	              // Calculate path choice
	              #tempRetValue := "LKinCtrl_CalcCircPathChoiceByIntermediatePointAndEndPoint"(circleStartPoint := #tempNextCmdIn.endPoint,
	                                                                                           circleEndPoint := #tempNextButOneCmdIn.endPoint,
	                                                                                           circleintermediatePoint := #tempNextButOneCmdIn.circleIntermediatePoint,
	                                                                                           pathPlane := #pathPlane,
	                                                                                           pathChoice => #tempNextButOneCmdIn.pathChoice);
	              
	              IF (#tempRetValue <> 0) THEN
	                #LKinCtrl_OffsetContour.returnValue := #tempRetValue;
	                #LKinCtrl_OffsetContour."region" := #COFF_REGION_TYPE_RAD_COMP_CIRC_CIRC;
	                #LKinCtrl_OffsetContour.subBlockNumber := 35058;
	                #LKinCtrl_OffsetContour.internalNumber := 431;
	                RETURN;
	              END_IF;
	              
	            ELSIF (#tempNextButOneCmdIn.circleMode = "CM_CENTER") THEN
	              // ------------ Via the circle center and the angle in a main plane ("CircMode" = 1) ------------
	              
	              // "Third" coordinate is ignored by system - also ignore here!
	              // Use start coordinate of circle instead
	              IF (#pathPlane = "CP_XZ") THEN
	                #tempNextButOneCmdIn.circleCenterPoint.y := #tempNextCmdIn.endPoint.y;
	              ELSIF (#pathPlane = "CP_YZ") THEN
	                #tempNextButOneCmdIn.circleCenterPoint.x := #tempNextCmdIn.endPoint.x;
	              ELSIF (#pathPlane = "CP_XY") THEN
	                #tempNextButOneCmdIn.circleCenterPoint.z := #tempNextCmdIn.endPoint.z;
	              END_IF;
	              
	              // Calculte correct circle end point - parameter not mandatory (and therefore probably not correct)
	              #tempRetValue := "LKinCtrl_CalcCircEndPointWithGivenCenterAndAngle"(circleStartPoint := #tempNextCmdIn.endPoint,
	                                                                                  circleCenterPoint := #tempNextButOneCmdIn.circleCenterPoint,
	                                                                                  pathPlane := #pathPlane,
	                                                                                  pathChoice := #tempNextButOneCmdIn.pathChoice,
	                                                                                  angle := #tempNextButOneCmdIn.circleAngle,
	                                                                                  endPoint => #tempNextButOneCmdIn.endPoint);
	              
	              IF (#tempRetValue <> 0) THEN
	                #LKinCtrl_OffsetContour.returnValue := #tempRetValue;
	                #LKinCtrl_OffsetContour."region" := #COFF_REGION_TYPE_RAD_COMP_CIRC_CIRC;
	                #LKinCtrl_OffsetContour.subBlockNumber := 35053;
	                #LKinCtrl_OffsetContour.internalNumber := 432;
	                RETURN;
	              END_IF;
	              
	            ELSIF (#tempNextButOneCmdIn.circleMode = "CM_RADIUS") THEN
	              // ------------ Via the circle radius and the end point in a main plane ("CircMode" = 2) ------------
	              #tempRetValue := "LKinCtrl_CalcCircCenterByRadiusAndEndPoint"(circleStartPoint := #tempNextCmdIn.endPoint,
	                                                                            circleEndPoint := #tempNextButOneCmdIn.endPoint,
	                                                                            pathPlane := #pathPlane,
	                                                                            circleRadius := #tempNextButOneCmdIn.circleRadius,
	                                                                            pathChoice := #tempNextButOneCmdIn.pathChoice,
	                                                                            circCenterPoint => #tempNextButOneCmdIn.circleCenterPoint);
	              
	              IF (#tempRetValue <> 0) THEN
	                #LKinCtrl_OffsetContour.returnValue := #tempRetValue;
	                #LKinCtrl_OffsetContour."region" := #COFF_REGION_TYPE_RAD_COMP_CIRC_CIRC;
	                #LKinCtrl_OffsetContour.subBlockNumber := 35052;
	                #LKinCtrl_OffsetContour.internalNumber := 433;
	                RETURN;
	              END_IF;
	              
	            END_IF;
	            
	            // Take care of next circular command
	            #tempRetValue := "LKinCtrl_CalcCircTangOrthPathPlane"(circlePoint := #tempNextCmdIn.endPoint,
	                                                                  circleCenterPoint := #tempNextButOneCmdIn.circleCenterPoint,
	                                                                  pathPlane := #pathPlane,
	                                                                  compDirection := #compensationDirection,
	                                                                  pathChoice := #tempNextButOneCmdIn.pathChoice,
	                                                                  vUnitTangentialPathPlane => #tempNextButOneCmdOut.tangentialUnitVecStart,
	                                                                  vUnitOrthogonalPathPlane => #tempNextButOneCmdOut.orthogonalUnitVecStart);
	            
	            IF (#tempRetValue <> 0) THEN
	              #LKinCtrl_OffsetContour.returnValue := #tempRetValue;
	              #LKinCtrl_OffsetContour."region" := #COFF_REGION_TYPE_RAD_COMP_CIRC_CIRC;
	              #LKinCtrl_OffsetContour.subBlockNumber := 35056;
	              #LKinCtrl_OffsetContour.internalNumber := 434;
	              RETURN;
	            END_IF;
	            
	            // Scale othogonal vector with tool radius to get orthogonal shift
	            #tempNextButOneCmdOut.orthogonalShiftStart := "LKinCtrl_VecScale"(vIn := #tempNextButOneCmdOut.orthogonalUnitVecStart,
	                                                                              factor := #toolRadius);
	            
	            
	            #tempNextButOneCmdOut.startPointOrthShifted := "LKinCtrl_VecAdd"(vIn1 := #tempNextCmdIn.endPoint,
	                                                                             vIn2 := #tempNextButOneCmdOut.orthogonalShiftStart);
	            
	            // ########## Intersection point of 1st circular and 2nd circular command  ##########
	            
	            IF (#tempNextCmdIn.circleMode = "CM_BORDER") THEN
	              // ------------ Via an intermediate point and the end point ("CircMode" = 0) ------------
	              // 3D circle possible
	              //
	              // Bring coordinates and parameters to same level as current point
	              #tempNextCmdStartPointOrhtShiftLevelled := #tempCurrentPointRadComp; //#tempNextCmdOut.startPointOrthShifted;
	              #tempNextCmdOut.circleCenterPoint := #tempNextCmdIn.circleCenterPoint;
	              
	              // Level parameters (third coordinate) with current point
	              CASE #pathPlane OF
	                "CP_XZ":
	                  #tempNextCmdStartPointOrhtShiftLevelled.y := #tempCurrentPoint.y;
	                  #tempNextCmdOut.circleCenterPoint.y := #tempCurrentPoint.y;
	                  
	                "CP_YZ":
	                  #tempNextCmdStartPointOrhtShiftLevelled.x := #tempCurrentPoint.x;
	                  #tempNextCmdOut.circleCenterPoint.x := #tempCurrentPoint.x;
	                  
	                "CP_XY":
	                  #tempNextCmdStartPointOrhtShiftLevelled.z := #tempCurrentPoint.z;
	                  #tempNextCmdOut.circleCenterPoint.z := #tempCurrentPoint.z;
	                ELSE
	                  #LKinCtrl_OffsetContour.returnValue := #ERR_COFF_INTERNAL;
	                  #LKinCtrl_OffsetContour."region" := #COFF_REGION_TYPE_RAD_COMP_CIRC_CIRC;
	                  #LKinCtrl_OffsetContour.internalNumber := 435;
	                  RETURN;
	              END_CASE;
	              
	              // Calculate radius of shifted 1st circle - levelled
	              #tempNextCmdOut.circleRadius := "LKinCtrl_VecAbs"("LKinCtrl_VecSub"(vIn1 := #tempNextCmdStartPointOrhtShiftLevelled,
	                                                                                                                                    vIn2 := #tempNextCmdOut.circleCenterPoint));
	            ELSE
	              #tempNextCmdOut.circleCenterPoint := #tempNextCmdIn.circleCenterPoint;
	              // Calculate radius of shifted 1st circle
	              #tempNextCmdOut.circleRadius := "LKinCtrl_VecAbs"("LKinCtrl_VecSub"(vIn1 := #tempCurrentPointRadComp,
	                                                                                                                                    vIn2 := #tempNextCmdOut.circleCenterPoint));
	            END_IF;
	            
	            IF (#tempNextButOneCmdIn.circleMode = "CM_BORDER") THEN
	              // ------------ Via an intermediate point and the end point ("CircMode" = 0) ------------
	              // 3D circle possible
	              //
	              // Bring coordinates and parameters to same level as current point
	              #tempNextButOneStartPointOrthShiftedLevelled := #tempNextButOneCmdOut.startPointOrthShifted;
	              #tempNextButOneCmdOut.circleCenterPoint := #tempNextButOneCmdIn.circleCenterPoint;
	              
	              // Level parameters (third coordinate) with current point
	              CASE #pathPlane OF
	                "CP_XZ":
	                  #tempNextButOneStartPointOrthShiftedLevelled.y := #tempCurrentPoint.y;
	                  #tempNextButOneCmdOut.circleCenterPoint.y := #tempCurrentPoint.y;
	                  
	                "CP_YZ":
	                  #tempNextButOneStartPointOrthShiftedLevelled.x := #tempCurrentPoint.x;
	                  #tempNextButOneCmdOut.circleCenterPoint.x := #tempCurrentPoint.x;
	                  
	                "CP_XY":
	                  #tempNextButOneStartPointOrthShiftedLevelled.z := #tempCurrentPoint.z;
	                  #tempNextButOneCmdOut.circleCenterPoint.z := #tempCurrentPoint.z;
	                ELSE
	                  #LKinCtrl_OffsetContour.returnValue := #ERR_COFF_INTERNAL;
	                  #LKinCtrl_OffsetContour."region" := #COFF_REGION_TYPE_RAD_COMP_CIRC_CIRC;
	                  #LKinCtrl_OffsetContour.internalNumber := 435;
	                  RETURN;
	              END_CASE;
	              // Calculate radius of shifted 2nd circle - levelled
	              #tempNextButOneCmdOut.circleRadius := "LKinCtrl_VecAbs"("LKinCtrl_VecSub"(vIn1 := #tempNextButOneStartPointOrthShiftedLevelled,
	                                                                                                                                                vIn2 := #tempNextButOneCmdOut.circleCenterPoint));
	            ELSE
	              #tempNextButOneCmdOut.circleCenterPoint := #tempNextButOneCmdIn.circleCenterPoint;
	              
	              // Calculate radius of shifted 2nd circle
	              // preliminary
	              #tempNextButOneCmdOut.circleRadius := "LKinCtrl_VecAbs"("LKinCtrl_VecSub"(vIn1 := #tempNextButOneCmdOut.startPointOrthShifted,
	                                                                                                                                                vIn2 := #tempNextButOneCmdOut.circleCenterPoint));
	            END_IF;
	            
	            // Intersection point of 1st and 2nd circle
	            #tempRetValue := "LKinCtrl_CalcCircleCircleIntersectionPoint"(circleCenterPoint1 := #tempNextCmdOut.circleCenterPoint,
	                                                                          circleCenterPoint2 := #tempNextButOneCmdOut.circleCenterPoint,
	                                                                          circleRadius1 := #tempNextCmdOut.circleRadius,
	                                                                          circleRadius2 := #tempNextButOneCmdOut.circleRadius,
	                                                                          pathPlane := #pathPlane,
	                                                                          intersectionPointA => #tempPa,
	                                                                          intersectionPointB => #tempPb);
	            IF (#tempRetValue <> 0) THEN
	              // V01.00.01
	              IF (#tempRetValue = #ERR_COFF_CIRCLE_CENTERS_EQUAL) THEN
	                // Circles are equal - use modified start point of following circle instead
	                #tempPa := #tempNextButOneCmdOut.startPointOrthShifted;
	                #tempPb := #tempNextButOneCmdOut.startPointOrthShifted;
	              ELSE
	                #LKinCtrl_OffsetContour.returnValue := #tempRetValue;
	                #LKinCtrl_OffsetContour."region" := #COFF_REGION_TYPE_RAD_COMP_CIRC_CIRC;
	                #LKinCtrl_OffsetContour.subBlockNumber := 35062;
	                #LKinCtrl_OffsetContour.internalNumber := 437;
	                RETURN;
	              END_IF;
	            END_IF;
	            
	            IF (#tempNextCmdIn.circleMode = "CM_BORDER") THEN
	              // ------------ Via an intermediate point and the end point ("CircMode" = 0) ------------
	              // 3D circle possible
	              // Relevel intersection point
	              CASE #pathPlane OF
	                "CP_XZ":
	                  #tempPa.y := #tempNextCmdIn.endPoint.y;
	                  #tempPb.y := #tempNextCmdIn.endPoint.y;
	                  
	                "CP_YZ":
	                  #tempPa.x := #tempNextCmdIn.endPoint.x;
	                  #tempPb.x := #tempNextCmdIn.endPoint.x;
	                  
	                "CP_XY":
	                  #tempPa.z := #tempNextCmdIn.endPoint.z;
	                  #tempPb.z := #tempNextCmdIn.endPoint.z;
	                ELSE
	                  #LKinCtrl_OffsetContour.returnValue := #ERR_COFF_INTERNAL;
	                  #LKinCtrl_OffsetContour."region" := #COFF_REGION_TYPE_RAD_COMP_CIRC_LIN;
	                  #LKinCtrl_OffsetContour.internalNumber := 436;
	                  RETURN;
	              END_CASE;
	            END_IF;
	            
	            // Two intersection points, use the one which is closer to the circle end point
	            #tempDistance1 := "LKinCtrl_VecAbs"("LKinCtrl_VecSub"(vIn1 := #tempNextCmdIn.endPoint, vIn2 := #tempPa));
	            #tempDistance2 := "LKinCtrl_VecAbs"("LKinCtrl_VecSub"(vIn1 := #tempNextCmdIn.endPoint, vIn2 := #tempPb));
	            
	            IF (#tempDistance1 < #tempDistance2) THEN
	              #tempNextCmdOut.endPoint := #tempPa;
	            ELSE
	              #tempNextCmdOut.endPoint := #tempPb;
	            END_IF;
	            
	          END_REGION
	          // ############# N E X T   B U T   O N E   C M D  -  N O N E #############
	        ELSE
	          REGION Next but one command NONE
	            // Output next but one coordinates - in case it's the last one
	            #tempNextButOneCmdOut.endPoint := #tempNextButOneCmdOut.endPointOrthShifted;
	            
	            // Calculate end point for circle (orthogonal shifted)
	            #tempRetValue := "LKinCtrl_CalcCircTangOrthPathPlane"(circlePoint := #tempNextCmdIn.endPoint,
	                                                                  circleCenterPoint := #tempNextCmdIn.circleCenterPoint,
	                                                                  pathPlane := #pathPlane,
	                                                                  compDirection := #compensationDirection,
	                                                                  pathChoice := #tempNextCmdIn.pathChoice,
	                                                                  vUnitTangentialPathPlane => #tempNextCmdOut.tangentialUnitVecEnd,
	                                                                  vUnitOrthogonalPathPlane => #tempNextCmdOut.orthogonalUnitVecEnd);
	            
	            IF (#tempRetValue <> 0) THEN
	              #LKinCtrl_OffsetContour.returnValue := #tempRetValue;
	              #LKinCtrl_OffsetContour."region" := #COFF_REGION_TYPE_RAD_COMP_CIRC_NONE;
	              #LKinCtrl_OffsetContour.subBlockNumber := 35056;
	              #LKinCtrl_OffsetContour.internalNumber := 450;
	              RETURN;
	            END_IF;
	            
	            // Scale othogonal vector with tool radius to get orthogonal shift
	            #tempNextCmdOut.orthogonalShiftEnd := "LKinCtrl_VecScale"(vIn := #tempNextCmdOut.orthogonalUnitVecEnd,
	                                                                      factor := #toolRadius);
	            
	            
	            #tempNextCmdOut.endPoint := "LKinCtrl_VecAdd"(vIn1 := #tempNextCmdIn.endPoint,
	                                                          vIn2 := #tempNextCmdOut.orthogonalShiftEnd);
	            (*
	            // Distinguish between different circular modes
	            IF (#tempNextCmdIn.circleMode = "CM_BORDER") THEN
	              // ------------ Via an intermediate point and the end point ("CircMode" = 0) ------------
	              
	              // Calculate end point for circle mode 0 by given mode 0
	              #tempRetValue := "LKinCtrl_CalcCircTangOrthPathPlane"(circlePoint := #tempNextCmdIn.endPoint,
	                                                                    circleCenterPoint := #tempNextCmdIn.circleCenterPoint,
	                                                                    pathPlane := #pathPlane,
	                                                                    compDirection := #compensationDirection,
	                                                                    pathChoice := #tempNextCmdIn.pathChoice,
	                                                                    vUnitTangentialPathPlane => #tempNextCmdOut.tangentialUnitVecEnd,
	                                                                    vUnitOrthogonalPathPlane => #tempNextCmdOut.orthogonalUnitVecEnd);
	              
	              IF (#tempRetValue <> 0) THEN
	                #LKinCtrl_OffsetContour.returnValue := #tempRetValue;
	                #LKinCtrl_OffsetContour."region" := #COFF_REGION_TYPE_RAD_COMP_CIRC_NONE;
	                #LKinCtrl_OffsetContour.subBlockNumber := 35056;
	                #LKinCtrl_OffsetContour.internalNumber := 450;
	                RETURN;
	              END_IF;
	              
	              // Scale othogonal vector with tool radius to get orthogonal shift
	              #tempNextCmdOut.orthogonalShiftEnd := "LKinCtrl_VecScale"(vIn := #tempNextCmdOut.orthogonalUnitVecEnd,
	                                                                        factor := #toolRadius);
	              
	              
	              #tempNextCmdOut.endPoint := "LKinCtrl_VecAdd"(vIn1 := #tempNextCmdIn.endPoint,
	                                                            vIn2 := #tempNextCmdOut.orthogonalShiftEnd);
	            ELSIF (#tempNextCmdIn.circleMode = "CM_CENTER") THEN
	              (*
	              // Calculate end point for circle mode 0 by given mode 1
	              #tempRetValue := "LKinCtrl_CalcCircEndPointWithGivenCenterAndAngle"(circleStartPoint := #tempCurrentPointRadComp,
	                                                                                  circleCenterPoint := #tempNextCmdIn.circleCenterPoint,
	                                                                                  pathPlane := #pathPlane,
	                                                                                  pathChoice := #tempNextCmdIn.pathChoice,
	                                                                                  angle := #tempNextCmdIn.circleAngle,
	                                                                                  endPoint => #tempNextCmdOut.endPoint);
	              
	              IF (#tempRetValue <> 0) THEN
	                #LKinCtrl_OffsetContour.returnValue := #tempRetValue;
	                #LKinCtrl_OffsetContour."region" := #COFF_REGION_TYPE_RAD_COMP_CIRC_NONE;
	                #LKinCtrl_OffsetContour.subBlockNumber := 35053;
	                #LKinCtrl_OffsetContour.internalNumber := 451;
	                RETURN;
	              END_IF;
	              *)
	              // Calculate end point for circle mode 0 by given mode 0
	              #tempRetValue := "LKinCtrl_CalcCircTangOrthPathPlane"(circlePoint := #tempNextCmdIn.endPoint,
	                                                                    circleCenterPoint := #tempNextCmdIn.circleCenterPoint,
	                                                                    pathPlane := #pathPlane,
	                                                                    compDirection := #compensationDirection,
	                                                                    pathChoice := #tempNextCmdIn.pathChoice,
	                                                                    vUnitTangentialPathPlane => #tempNextCmdOut.tangentialUnitVecEnd,
	                                                                    vUnitOrthogonalPathPlane => #tempNextCmdOut.orthogonalUnitVecEnd);
	              
	              IF (#tempRetValue <> 0) THEN
	                #LKinCtrl_OffsetContour.returnValue := #tempRetValue;
	                #LKinCtrl_OffsetContour."region" := #COFF_REGION_TYPE_RAD_COMP_CIRC_NONE;
	                #LKinCtrl_OffsetContour.subBlockNumber := 35056;
	                #LKinCtrl_OffsetContour.internalNumber := 450;
	                RETURN;
	              END_IF;
	              
	              // Scale othogonal vector with tool radius to get orthogonal shift
	              #tempNextCmdOut.orthogonalShiftEnd := "LKinCtrl_VecScale"(vIn := #tempNextCmdOut.orthogonalUnitVecEnd,
	                                                                        factor := #toolRadius);
	              
	              
	              #tempNextCmdOut.endPoint := "LKinCtrl_VecAdd"(vIn1 := #tempNextCmdIn.endPoint,
	                                                            vIn2 := #tempNextCmdOut.orthogonalShiftEnd);
	              
	            ELSIF (#tempNextCmdIn.circleMode = "CM_RADIUS") THEN
	              (*
	              // ------------ Via the circle radius and the end point in a main plane ("CircMode" = 2) ------------
	              // Calculate angle between center/start and center/end of circle - always the smaller one!!!
	              #tempRetValue := "LKinCtrl_CalcAngleBetweenVectors"(point1 := #tempCurrentPointRadComp,//#tempNextCmdOut.startPointOrthShifted,
	                                                                  point2 := #tempNextCmdIn.endPoint,//#tempNextCmdOut.endPoint,
	                                                                  intersectionPoint := #tempNextCmdIn.circleCenterPoint,
	                                                                  angle => #tempAngle);
	              
	              IF (#tempRetValue <> 0) THEN
	                #LKinCtrl_OffsetContour.returnValue := #tempRetValue;
	                #LKinCtrl_OffsetContour."region" := #COFF_REGION_TYPE_RAD_COMP_CIRC_NONE;
	                #LKinCtrl_OffsetContour.subBlockNumber := 35059;
	                #LKinCtrl_OffsetContour.internalNumber := 452;
	                RETURN;
	              END_IF;
	              
	              // Calculate end point for circle mode 0 by given mode 2
	              #tempRetValue := "LKinCtrl_CalcCircEndPointWithGivenCenterAndAngle"(circleStartPoint := #tempCurrentPointRadComp, //tempNextCmdOut.startPointOrthShifted,
	                                                                                  circleCenterPoint := #tempNextCmdIn.circleCenterPoint,
	                                                                                  pathPlane := #pathPlane,
	                                                                                  pathChoice := #tempNextCmdIn.pathChoice,
	                                                                                  angle := #tempAngle,
	                                                                                  endPoint => #tempNextCmdOut.endPoint);
	              
	              
	              
	              IF (#tempRetValue <> 0) THEN
	                #LKinCtrl_OffsetContour.returnValue := #tempRetValue;
	                #LKinCtrl_OffsetContour."region" := #COFF_REGION_TYPE_RAD_COMP_CIRC_NONE;
	                #LKinCtrl_OffsetContour.subBlockNumber := 35053;
	                #LKinCtrl_OffsetContour.internalNumber := 453;
	                RETURN;
	              END_IF;
	              *)
	              ;
	            END_IF;
	            *)
	            
	          END_REGION
	        END_IF;
	        
	        
	        // ############# M O D I F Y   N E X T   C I R C U L A R   C O M M A N D   #############
	        REGION Modify next circular command
	          // Distinguish between different circular modes
	          IF (#tempNextCmdIn.circleMode = "CM_BORDER") THEN
	            
	            // ------------ Via an intermediate point and the end point ("CircMode" = 0) ------------
	            // Calculate intermediate point for circle mode 0 by given mode 0
	            // Calculate circle paramters
	            #tempRetValue := "LKinCtrl_CalcCircTangOrthPathPlane"(circlePoint := #tempNextCmdIn.circleIntermediatePoint,
	                                                                  circleCenterPoint := #tempNextCmdIn.circleCenterPoint,
	                                                                  pathPlane := #pathPlane,
	                                                                  compDirection := #compensationDirection,
	                                                                  pathChoice := #tempNextCmdIn.pathChoice,
	                                                                  vUnitTangentialPathPlane => #tempNextCmdOut.tangentialUnitVecIntermediate,
	                                                                  vUnitOrthogonalPathPlane => #tempNextCmdOut.orthogonalUnitVecIntermediate);
	            
	            IF (#tempRetValue <> 0) THEN
	              #LKinCtrl_OffsetContour.returnValue := #tempRetValue;
	              #LKinCtrl_OffsetContour."region" := #COFF_REGION_TYPE_RAD_COMP_CIRC_GEN;
	              #LKinCtrl_OffsetContour.subBlockNumber := 35056;
	              #LKinCtrl_OffsetContour.internalNumber := 460;
	              RETURN;
	            END_IF;
	            
	            // Scale othogonal vector with tool radius to get orthogonal shift
	            #tempNextCmdOut.orthogonalShiftIntermediate := "LKinCtrl_VecScale"(vIn := #tempNextCmdOut.orthogonalUnitVecIntermediate,
	                                                                               factor := #toolRadius);
	            
	            
	            #tempNextCmdOut.circleIntermediatePoint := "LKinCtrl_VecAdd"(vIn1 := #tempNextCmdIn.circleIntermediatePoint,
	                                                                         vIn2 := #tempNextCmdOut.orthogonalShiftIntermediate);
	            
	            // Change circle mode to 0 - intermediate point and the end point ("CircMode" = 0)
	            #tempNextCmdOut.circleMode := "CM_BORDER";
	            
	          ELSIF (#tempNextCmdIn.circleMode = "CM_CENTER") THEN
	            
	            // Take care of greater angles
	            // #tempMod := TRUNC(#tempNextCmdIn.circleAngle / 180.0);
	            // IF (#tempMod >= 3) THEN
	            //   #tempAngle := #tempNextCmdIn.circleAngle - ((#tempMod - 1) * 180);
	            // ELSE
	            //   #tempAngle := #tempNextCmdIn.circleAngle;
	            // END_IF;
	            
	            // V01.02.02
	            // Calculate compensated angle
	            #tempRetValue := "LKinCtrl_CalcAngleBetweenVectors"(point1 := #tempCurrentPointRadComp, //tempNextCmdOut.startPointOrthShifted,
	                                                                point2 := #tempNextCmdOut.endPoint,
	                                                                intersectionPoint := #tempNextCmdIn.circleCenterPoint,
	                                                                angle => #tempAngle);
	            
	            IF (#tempRetValue <> 0) THEN
	              #LKinCtrl_OffsetContour.returnValue := #tempRetValue;
	              #LKinCtrl_OffsetContour."region" := #COFF_REGION_TYPE_RAD_COMP_CIRC_GEN;
	              #LKinCtrl_OffsetContour.subBlockNumber := 35059;
	              #LKinCtrl_OffsetContour.internalNumber := 461;
	              RETURN;
	            END_IF;
	            //
	            // Calculate intermediate point for circle mode 0 by given mode 1
	            #tempRetValue := "LKinCtrl_CalcCircEndPointWithGivenCenterAndAngle"(circleStartPoint := #tempCurrentPointRadComp, // tempNextCmdOut.startPointOrthShifted,
	                                                                                circleCenterPoint := #tempNextCmdIn.circleCenterPoint,
	                                                                                pathPlane := #pathPlane,
	                                                                                pathChoice := #tempNextCmdIn.pathChoice,
	                                                                                angle := #tempAngle / 2.0,//(#tempNextCmdIn.circleAngle / 2.0),
	                                                                                endPoint => #tempNextCmdOut.circleIntermediatePoint);
	            IF (#tempRetValue <> 0) THEN
	              #LKinCtrl_OffsetContour.returnValue := #tempRetValue;
	              #LKinCtrl_OffsetContour."region" := #COFF_REGION_TYPE_RAD_COMP_CIRC_GEN;
	              #LKinCtrl_OffsetContour.subBlockNumber := 35053;
	              #LKinCtrl_OffsetContour.internalNumber := 462;
	              RETURN;
	            END_IF;
	            
	            // Ceck if resulting path choice (circle with intermediate point) has changed --> circle larger than 360°
	            // Calculate path choice
	            #tempRetValue := "LKinCtrl_CalcCircPathChoiceByIntermediatePointAndEndPoint"(circleStartPoint := #tempCurrentPointRadComp, //tempNextCmdOut.startPointOrthShifted,
	                                                                                         circleEndPoint := #tempNextCmdOut.endPoint,
	                                                                                         circleintermediatePoint := #tempNextCmdOut.circleIntermediatePoint,
	                                                                                         pathPlane := #pathPlane,
	                                                                                         pathChoice => #tempPathChoice);
	            
	            
	            IF (#tempRetValue <> 0) THEN
	              #LKinCtrl_OffsetContour.returnValue := #tempRetValue;
	              #LKinCtrl_OffsetContour."region" := #COFF_REGION_TYPE_RAD_COMP_CIRC_GEN;
	              #LKinCtrl_OffsetContour.subBlockNumber := 35058;
	              #LKinCtrl_OffsetContour.internalNumber := 463;
	              RETURN;
	            END_IF;
	            
	            IF ((#tempNextCmdIn.pathChoice <> #tempPathChoice) OR
	              (#tempNextCmdIn.circleAngle >= 360.0))
	            THEN
	              
	              // V01.02.02 - done before now
	              // // Calculate additional angle between center/start and center/end of circle - always the smaller one!!!
	              // #tempRetValue := "LKinCtrl_CalcAngleBetweenVectors"(point1 := #tempCurrentPointRadComp, //tempNextCmdOut.startPointOrthShifted,
	              //                                                     point2 := #tempNextCmdOut.endPoint,
	              //                                                     intersectionPoint := #tempNextCmdIn.circleCenterPoint,
	              //                                                     angle => #tempAngle);
	              
	              // IF (#tempRetValue <> 0) THEN
	              //   #LKinCtrl_OffsetContour.returnValue := #tempRetValue;
	              //   #LKinCtrl_OffsetContour."region" := #COFF_REGION_TYPE_RAD_COMP_CIRC_GEN;
	              //   #LKinCtrl_OffsetContour.subBlockNumber := 35059;
	              //   #LKinCtrl_OffsetContour.internalNumber := 463;
	              //   RETURN;
	              // END_IF;
	              
	              // Circle > 360° - not possible with circle type border
	              IF (#tempNextCmdIn.pathChoice <> #tempPathChoice) THEN
	                #tempNextCmdOut.circleAngle := (TRUNC((#tempNextCmdIn.circleAngle + 180.0) / 360.0) * 360.0) + #tempAngle;
	              ELSE
	                #tempNextCmdOut.circleAngle := (TRUNC((#tempNextCmdIn.circleAngle + 180.0) / 360.0) * 360.0) - #tempAngle;
	              END_IF;
	              
	              #tempNextCmdOut.circleMode := "CM_CENTER";
	            ELSE
	              
	              // V01.02.02
	              // Output angle - for debugging only
	              #tempNextCmdOut.circleAngle := #tempAngle;
	              
	              // Change circle mode to 0 - intermediate point and the end point ("CircMode" = 0)
	              #tempNextCmdOut.circleMode := "CM_BORDER";
	            END_IF;
	            
	          ELSIF (#tempNextCmdIn.circleMode = "CM_RADIUS") THEN
	            // ------------ Via the circle radius and the end point in a main plane ("CircMode" = 2) ------------
	            // Calculate angle between center/start and center/end of circle - always the smaller one!!!
	            #tempRetValue := "LKinCtrl_CalcAngleBetweenVectors"(point1 := #tempCurrentPointRadComp,
	                                                                point2 := #tempNextCmdOut.endPoint,
	                                                                intersectionPoint := #tempNextCmdIn.circleCenterPoint,
	                                                                angle => #tempAngle);
	            
	            IF (#tempRetValue <> 0) THEN
	              #LKinCtrl_OffsetContour.returnValue := #tempRetValue;
	              #LKinCtrl_OffsetContour."region" := #COFF_REGION_TYPE_RAD_COMP_CIRC_GEN;
	              #LKinCtrl_OffsetContour.subBlockNumber := 35059;
	              #LKinCtrl_OffsetContour.internalNumber := 464;
	              RETURN;
	            END_IF;
	            
	            // Calculate intermediate point for circle mode 0 by given mode 2
	            #tempRetValue := "LKinCtrl_CalcCircEndPointWithGivenCenterAndAngle"(circleStartPoint := #tempCurrentPointRadComp, //tempNextCmdOut.startPointOrthShifted,
	                                                                                circleCenterPoint := #tempNextCmdIn.circleCenterPoint,
	                                                                                pathPlane := #pathPlane,
	                                                                                pathChoice := #tempNextCmdIn.pathChoice,
	                                                                                angle := (#tempAngle / 2.0),
	                                                                                endPoint => #tempNextCmdOut.circleIntermediatePoint);
	            
	            IF (#tempRetValue <> 0) THEN
	              #LKinCtrl_OffsetContour.returnValue := #tempRetValue;
	              #LKinCtrl_OffsetContour."region" := #COFF_REGION_TYPE_RAD_COMP_CIRC_GEN;
	              #LKinCtrl_OffsetContour.subBlockNumber := 35053;
	              #LKinCtrl_OffsetContour.internalNumber := 465;
	              RETURN;
	            END_IF;
	            
	            // Change circle mode to 0 - intermediate point and the end point ("CircMode" = 0)
	            #tempNextCmdOut.circleMode := "CM_BORDER";
	            
	          END_IF;
	          
	          // Additional check - has the direction between start - end and start - compensated end changed
	          // --> Reversal path with "small" length (and "large" tool radius) leads to unexpected circle (mathematical correct but in an unexpected direction)
	          REGION Additional plausibility check
	            #tempRetValue := "LKinCtrl_CalcAngleBetweenVectors"(point1 := #tempNextCmdOut.endPoint,
	                                                                point2 := #tempNextCmdIn.endPoint,
	                                                                intersectionPoint := #tempCurrentPoint,
	                                                                angle => #tempAngle);
	            
	            IF (#tempRetValue <> 0) THEN
	              #LKinCtrl_OffsetContour.returnValue := #tempRetValue;
	              #LKinCtrl_OffsetContour."region" := #COFF_REGION_TYPE_RAD_COMP_CIRC_GEN;
	              #LKinCtrl_OffsetContour.subBlockNumber := 35059;
	              #LKinCtrl_OffsetContour.internalNumber := 470;
	              RETURN;
	            END_IF;
	            
	            IF ((#tempAngle > #COFF_CIRC_REVERSAL_TOLERANCE_ANGLE) AND
	              ("LKinCtrl_VecAbs"("LKinCtrl_VecSub"(vIn1 := #tempNextCmdOut.endPoint,
	                                                                      vIn2 := #tempNextCmdOut.circleIntermediatePoint)) < (2.0 * #toolRadius)))
	            THEN
	              #LKinCtrl_OffsetContour.returnValue := #ERR_COFF_NO_SOLUTION_FOR_GIVEN_CIRCULAR_CMD;
	              #LKinCtrl_OffsetContour."region" := #COFF_REGION_TYPE_RAD_COMP_CIRC_GEN;
	              #LKinCtrl_OffsetContour.subBlockNumber := 0;
	              #LKinCtrl_OffsetContour.internalNumber := 471;
	              RETURN;
	            END_IF;
	            
	          END_REGION
	          
	          // V01.02.02
	          REGION Additional plausibility check
	            // Check if circle radius has become smaller than possible - compensation inside
	            
	            // Calculate the length end point circle center 
	            #tempRetValue := "LKinCtrl_CalcVecDistancePathPlane"(vectorInA := #tempNextCmdIn.endPoint,
	                                                                 vectorInB := #tempNextCmdIn.circleCenterPoint,
	                                                                 pathPlane := #pathPlane,
	                                                                 distancePathPlane => #tempCircleDistance1);
	            
	            IF (#tempRetValue <> 0) THEN
	              #LKinCtrl_OffsetContour.returnValue := #tempRetValue;
	              #LKinCtrl_OffsetContour."region" := #COFF_REGION_TYPE_RAD_COMP_CIRC_GEN;
	              #LKinCtrl_OffsetContour.subBlockNumber := 35067;
	              #LKinCtrl_OffsetContour.internalNumber := 472;
	              RETURN;
	            END_IF;
	            
	            #tempRetValue := "LKinCtrl_CalcVecDistancePathPlane"(vectorInA := #tempNextCmdOut.endPoint,
	                                                                 vectorInB := #tempNextCmdIn.circleCenterPoint,
	                                                                 pathPlane := #pathPlane,
	                                                                 distancePathPlane => #tempCircleDistance2);
	            
	            IF (#tempRetValue <> 0) THEN
	              #LKinCtrl_OffsetContour.returnValue := #tempRetValue;
	              #LKinCtrl_OffsetContour."region" := #COFF_REGION_TYPE_RAD_COMP_CIRC_GEN;
	              #LKinCtrl_OffsetContour.subBlockNumber := 35067;
	              #LKinCtrl_OffsetContour.internalNumber := 473;
	              RETURN;
	            END_IF;
	            
	            IF (#tempCircleDistance2 < #tempCircleDistance1) THEN
	              // inside circle - check plausibility
	              // Tool radius must not be greater than circle radius
	              IF (#toolRadius > (#tempCircleDistance1 - #RADIUS_PLAUSIBLITY_TOLERANCE)) THEN
	                #LKinCtrl_OffsetContour.returnValue := #ERR_COFF_NO_SOLUTION_FOR_GIVEN_CIRCULAR_CMD;
	                #LKinCtrl_OffsetContour."region" := #COFF_REGION_TYPE_RAD_COMP_CIRC_GEN;
	                #LKinCtrl_OffsetContour.subBlockNumber := 0;
	                #LKinCtrl_OffsetContour.internalNumber := 474;
	                RETURN;
	              END_IF;
	              // Tool radius must not be greater than circle start and end point (uncompensated)
	              #tempRetValue := "LKinCtrl_CalcVecDistancePathPlane"(vectorInA := #tempCurrentPoint,
	                                                                   vectorInB := #tempNextCmdIn.endPoint,
	                                                                   pathPlane := #pathPlane,
	                                                                   distancePathPlane => #tempCircleDistance3);
	              
	              IF (#tempRetValue <> 0) THEN
	                #LKinCtrl_OffsetContour.returnValue := #tempRetValue;
	                #LKinCtrl_OffsetContour."region" := #COFF_REGION_TYPE_RAD_COMP_CIRC_GEN;
	                #LKinCtrl_OffsetContour.subBlockNumber := 35067;
	                #LKinCtrl_OffsetContour.internalNumber := 475;
	                RETURN;
	              END_IF;
	              
	              IF (#toolRadius > (#tempCircleDistance3 - #RADIUS_PLAUSIBLITY_TOLERANCE)) THEN
	                #LKinCtrl_OffsetContour.returnValue := #ERR_COFF_NO_SOLUTION_FOR_GIVEN_CIRCULAR_CMD;
	                #LKinCtrl_OffsetContour."region" := #COFF_REGION_TYPE_RAD_COMP_CIRC_GEN;
	                #LKinCtrl_OffsetContour.subBlockNumber := 0;
	                #LKinCtrl_OffsetContour.internalNumber := 476;
	                RETURN;
	              END_IF;
	              
	            END_IF;
	            
	          END_REGION
	        END_REGION
	      END_IF;
	    END_REGION
	    
	  END_IF;
	  
	  // V01.00.01
	  // Output before length compensation
	  #nextPositionAbsoluteRadCompOut := "LKinCtrl_3DPointToCartesianCoord"(#tempNextCmdOut.endPoint);
	END_REGION TOOL_RADIUS_COMPENSATION
	
	// Tool length compensation
	REGION TOOL_LENGTH_COMPENSATION
	  IF (#tempToolLengthComp) THEN
	    // Next command
	    // -------------------------------------------------------------------------------------
	    // Compensate coordinates of according to path plane
	    // End point
	    #tempRetValue := "LKinCtrl_CalcToolLengthCompensation"(toolLength := #toolLength,
	                                                           pathPlane := #pathPlane,
	                                                           point := #tempNextCmdOut.endPoint);
	    IF (#tempRetValue <> 0) THEN
	      #LKinCtrl_OffsetContour.returnValue := #tempRetValue;
	      #LKinCtrl_OffsetContour."region" := #COFF_REGION_TYPE_LEN_COMP_NEXT;
	      #LKinCtrl_OffsetContour.subBlockNumber := 35070;
	      #LKinCtrl_OffsetContour.internalNumber := 601;
	      RETURN;
	    END_IF;
	    
	    // Circle coordinates
	    IF (#tempNextCmdOut.cmdType = "LKINCTRL_MC_MOVECIRCULARABS") THEN
	      
	      IF (#tempNextCmdOut.circleMode = "CM_BORDER") THEN
	        
	        #tempRetValue := "LKinCtrl_CalcToolLengthCompensation"(toolLength := #toolLength,
	                                                               pathPlane := #pathPlane,
	                                                               point := #tempNextCmdOut.circleIntermediatePoint);
	        IF (#tempRetValue <> 0) THEN
	          #LKinCtrl_OffsetContour.returnValue := #tempRetValue;
	          #LKinCtrl_OffsetContour."region" := #COFF_REGION_TYPE_LEN_COMP_NEXT;
	          #LKinCtrl_OffsetContour.subBlockNumber := 35070;
	          #LKinCtrl_OffsetContour.internalNumber := 602;
	          RETURN;
	        END_IF;
	        
	      ELSIF (#tempNextCmdOut.circleMode = "CM_CENTER") THEN
	        
	        #tempRetValue := "LKinCtrl_CalcToolLengthCompensation"(toolLength := #toolLength,
	                                                               pathPlane := #pathPlane,
	                                                               point := #tempNextCmdOut.circleCenterPoint);
	        IF (#tempRetValue <> 0) THEN
	          #LKinCtrl_OffsetContour.returnValue := #tempRetValue;
	          #LKinCtrl_OffsetContour."region" := #COFF_REGION_TYPE_LEN_COMP_NEXT;
	          #LKinCtrl_OffsetContour.subBlockNumber := 35070;
	          #LKinCtrl_OffsetContour.internalNumber := 603;
	          RETURN;
	        END_IF;
	        
	      ELSIF (#tempNextCmdOut.circleMode = "CM_RADIUS") THEN
	        ;
	      ELSE
	        #LKinCtrl_OffsetContour.returnValue := #ERR_COFF_INTERNAL; // Internal error
	        #LKinCtrl_OffsetContour."region" := #COFF_REGION_TYPE_LEN_COMP_NEXT;
	        #LKinCtrl_OffsetContour.internalNumber := 604;
	        RETURN;
	      END_IF;
	    END_IF;
	    
	    // Intermediate command
	    // -------------------------------------------------------------------------------------
	    // Compensate coordinates of according to path plane
	    IF (#tempIntermediateCmdOut.cmdType <> -1) THEN
	      
	      // End point
	      #tempRetValue := "LKinCtrl_CalcToolLengthCompensation"(toolLength := #toolLength,
	                                                             pathPlane := #pathPlane,
	                                                             point := #tempIntermediateCmdOut.endPoint);
	      IF (#tempRetValue <> 0) THEN
	        #LKinCtrl_OffsetContour.returnValue := #tempRetValue;
	        #LKinCtrl_OffsetContour."region" := #COFF_REGION_TYPE_LEN_COMP_INTER_CMD;
	        #LKinCtrl_OffsetContour.subBlockNumber := 35070;
	        #LKinCtrl_OffsetContour.internalNumber := 605;
	        RETURN;
	      END_IF;
	      
	      // Always circle by intemdiate point and end point
	      #tempRetValue := "LKinCtrl_CalcToolLengthCompensation"(toolLength := #toolLength,
	                                                             pathPlane := #pathPlane,
	                                                             point := #tempIntermediateCmdOut.circleIntermediatePoint);
	      IF (#tempRetValue <> 0) THEN
	        #LKinCtrl_OffsetContour.returnValue := #tempRetValue;
	        #LKinCtrl_OffsetContour."region" := #COFF_REGION_TYPE_LEN_COMP_INTER_CMD;
	        #LKinCtrl_OffsetContour.subBlockNumber := 35070;
	        #LKinCtrl_OffsetContour.internalNumber := 606;
	        RETURN;
	      END_IF;
	    END_IF;
	    
	    // Next but one command - not needed - no output
	    // -------------------------------------------------------------------------------------
	    (*
	    // Compensate coordinates of according to path plane
	    // End point
	    #tempRetValue := "LKinCtrl_CalcToolLengthCompensation"(toolLength := #toolLength,
	                                                           pathPlane := #pathPlane,
	                                                           point := #tempNextButOneCmdOut.endPoint);
	    IF (#tempRetValue <> 0) THEN
	      #LKinCtrl_OffsetContour.returnValue := #tempRetValue;
	      #LKinCtrl_OffsetContour."region" := #COFF_REGION_TYPE_LEN_COMP_NEXT_BUT_ONE_CMD;
	      #LKinCtrl_OffsetContour.subBlockNumber := 35070;
	      #LKinCtrl_OffsetContour.internalNumber := 607
	      RETURN;
	    END_IF;
	    *)
	  END_IF;
	END_REGION
	
	REGION Output data
	  
	  // ############# O U T P U T   D A T A  #############
	  // ###################################### 
	  IF (#tempToolRadiusComp OR #tempToolLengthComp) THEN
	    // Next command
	    
	    #nextCommandOut.cmdType := #tempNextCmdOut.cmdType;
	    #nextCommandOut.cmdCoordinates.cartesianPosition := "LKinCtrl_3DPointToCartesianCoord"(#tempNextCmdOut.endPoint);
	    
	    IF (#tempNextCmdOut.cmdType = "LKINCTRL_MC_MOVECIRCULARABS") THEN
	      #nextCommandOut.cmdParameters.circleParameters.circMode := #tempNextCmdOut.circleMode;
	      
	      IF (#tempNextCmdOut.circleMode = "CM_BORDER") THEN
	        #nextCommandOut.cmdParameters.circleParameters.auxPoint[1] := #tempNextCmdOut.circleIntermediatePoint.x;
	        #nextCommandOut.cmdParameters.circleParameters.auxPoint[2] := #tempNextCmdOut.circleIntermediatePoint.y;
	        #nextCommandOut.cmdParameters.circleParameters.auxPoint[3] := #tempNextCmdOut.circleIntermediatePoint.z;
	        // *** AW 2022-05-29 - debugging only - compensated angle
	        #nextCommandOut.cmdParameters.circleParameters.arc := #tempNextCmdOut.circleAngle;
	        
	      ELSIF (#tempNextCmdOut.circleMode = "CM_CENTER") THEN
	        #nextCommandOut.cmdParameters.circleParameters.pathChoice := #tempNextCmdIn.pathChoice;
	        #nextCommandOut.cmdParameters.circleParameters.circlePlane := #tempNextCmdIn.circlePlane;
	        #nextCommandOut.cmdParameters.circleParameters.auxPoint[1] := #tempNextCmdOut.circleCenterPoint.x;
	        #nextCommandOut.cmdParameters.circleParameters.auxPoint[2] := #tempNextCmdOut.circleCenterPoint.y;
	        #nextCommandOut.cmdParameters.circleParameters.auxPoint[3] := #tempNextCmdOut.circleCenterPoint.z;
	        #nextCommandOut.cmdParameters.circleParameters.arc := #tempNextCmdOut.circleAngle; // #tempNextCmdIn.circleAngle;
	        
	      ELSIF (#tempNextCmdOut.circleMode = "CM_RADIUS") THEN
	        #nextCommandOut.cmdParameters.circleParameters.pathChoice := #tempNextCmdIn.pathChoice;
	        #nextCommandOut.cmdParameters.circleParameters.circlePlane := #tempNextCmdIn.circlePlane;
	        #nextCommandOut.cmdParameters.circleParameters.radius := #tempNextCmdIn.circleRadius;
	        
	      ELSE
	        #LKinCtrl_OffsetContour.returnValue := #ERR_COFF_INTERNAL; // Internal error
	        #LKinCtrl_OffsetContour."region" := #COFF_REGION_TYPE_OUTPUT_DATA;
	        RETURN;
	      END_IF;
	    END_IF;
	    
	    // Coordinate a
	    // ------------
	    // Linear absolute
	    IF (#tempNextCmdIn.cmdType = "LKINCTRL_MC_MOVELINEARABS") THEN
	      // Absolute coordinates
	      #nextCommandOut.cmdCoordinates.cartesianPosition.a := #nextCommandIn.cmdCoordinates.cartesianPosition.a;
	      // Linear relative
	    ELSIF (#tempNextCmdIn.cmdType = "LKINCTRL_MC_MOVELINEARREL") THEN
	      // Relative coordinates -> calculate absolute coordinate (always)
	      #nextCommandOut.cmdCoordinates.cartesianPosition.a := #currentPosIn.positionAbsolute.a + #nextCommandIn.cmdCoordinates.cartesianPosition.a;
	      // Circular absolute  
	    ELSIF (#tempNextCmdIn.cmdType = "LKINCTRL_MC_MOVECIRCULARABS") THEN
	      // Absolute coordinates
	      #nextCommandOut.cmdCoordinates.cartesianPosition.a := #nextCommandIn.cmdCoordinates.cartesianPosition.a;
	      // Circular relative  
	    ELSIF (#tempNextCmdIn.cmdType = "LKINCTRL_MC_MOVECIRCULARREL") THEN
	      // Relative coordinates -> calculate absolute coordinate (always)
	      #nextCommandOut.cmdCoordinates.cartesianPosition.a := #currentPosIn.positionAbsolute.a + #nextCommandIn.cmdCoordinates.cartesianPosition.a;
	    END_IF;
	    
	    // Output absolute end point for next cycle (including coordinate a)
	    #nextPositionAbsoluteOut := "LKinCtrl_3DPointToCartesianCoord"(#tempNextCmdIn.endPoint);
	    #nextPositionAbsoluteOut.a := #nextCommandOut.cmdCoordinates.cartesianPosition.a;
	    
	    // Output absolute end point (radius compensated) for next cycle (including coordinate a)
	    // V01.00.01
	    // nextPositionAbsoluteRadCompOut := "LKinCtrl_3DPointToCartesianCoord"(#tempNextCmdOut.endPoint);
	    #nextPositionAbsoluteRadCompOut.a := #nextCommandOut.cmdCoordinates.cartesianPosition.a;
	    
	    // Intermediate command
	    IF (#tempIntermediateCmdOut.cmdType <> -1) THEN
	      
	      // Take all parameter preliminary
	      #intermediateCommandOut := #nextCommandIn;
	      
	      #intermediateCommandOut.cmdType := #tempIntermediateCmdOut.cmdType;
	      #intermediateCommandOut.cmdParameters.circleParameters.circMode := #tempIntermediateCmdOut.circleMode;
	      
	      // Circle by intemdiate point and end point
	      #intermediateCommandOut.cmdCoordinates.cartesianPosition := "LKinCtrl_3DPointToCartesianCoord"(#tempIntermediateCmdOut.endPoint);
	      #intermediateCommandOut.cmdParameters.circleParameters.auxPoint[1] := #tempIntermediateCmdOut.circleIntermediatePoint.x;
	      #intermediateCommandOut.cmdParameters.circleParameters.auxPoint[2] := #tempIntermediateCmdOut.circleIntermediatePoint.y;
	      #intermediateCommandOut.cmdParameters.circleParameters.auxPoint[3] := #tempIntermediateCmdOut.circleIntermediatePoint.z;
	      
	      // Coordinate a
	      #intermediateCommandOut.cmdCoordinates.cartesianPosition.a := #nextCommandOut.cmdCoordinates.cartesianPosition.a;
	    ELSE
	      #intermediateCommandOut.cmdType := -1;
	    END_IF;
	    
	    // Next but one command
	    //nextButOneCommandOut.cmdType := #tempNextButOneCmdIn.cmdType;
	    //nextButOneCommandOut.cmdCoordinates.cartesianPosition := "LKinCtrl_3DPointToCartesianCoord"(#tempNextButOneCmdOut.endPoint);
	    #nextButOneCommandOut.transitionParameter[1] := #tempNextButOneCmdOut.transitionParameter1;
	  ELSE
	    // Next command
	    #nextCommandOut := #nextCommandIn;
	  END_IF;
	  
	END_REGION
	
	#LKinCtrl_OffsetContour.returnValue := 16#0;
	#LKinCtrl_OffsetContour."region" := #COFF_REGION_TYPE_NONE;
	#LKinCtrl_OffsetContour.subBlockNumber := 16#0;
	#LKinCtrl_OffsetContour.internalNumber := 0;
	
	
END_FUNCTION

FUNCTION "LKinCtrl_CartesianCoordTo3DPoint" : "LKinCtrl_typeCOff3DPoint"
TITLE = LKinCtrl_CartesianCoordTo3DPoint
{ S7_Optimized_Access := 'TRUE' }
AUTHOR : 'handling.team.automation@siemens.com'
FAMILY : LKinCtrl
VERSION : 5.0
//The function converts data type "LKinCtrl_typeCartesianPosition" in "LKinCtrl_typeCOff3DPoint"
   VAR_INPUT 
      cartesianCoord : "LKinCtrl_typeCartesianPosition";   // Cartesian input coordinate
   END_VAR


BEGIN
	//==========================================================================================
	// SIEMENS AG
	// (c)Copyright 2019 All Rights Reserved
	//------------------------------------------------------------------------------------------
	// Library: LCOffset
	// Tested with: S7-1515T-3 PN/DP
	// Engineering: TIA Portal V15
	// Restrictions: ---
	// Requirements: S7-1500T FW 2.5
	// Functionality: The function converts data type "LKinCtrl_typeCartesianPosition" in "LKinCtrl_typeCOff3DPoint"
	// Support: tech.team.motioncontrol@siemens.com
	// Note: Parameter comments are only available in language 'English (United States)'
	//------------------------------------------------------------------------------------------
	// Change log table:
	// Version    Date          Expert in charge    Changes applied
	// 01.00.00   2019-02-14    AW                  created
	//===========================================================================================
	//
	#LKinCtrl_CartesianCoordTo3DPoint.x := #cartesianCoord.x;
	#LKinCtrl_CartesianCoordTo3DPoint.y := #cartesianCoord.y;
	#LKinCtrl_CartesianCoordTo3DPoint.z := #cartesianCoord.z;
END_FUNCTION

FUNCTION "LKinCtrl_VecAdd" : "LKinCtrl_typeCOff3DPoint"
TITLE = LKinCtrl_VecAdd
{ S7_Optimized_Access := 'TRUE' }
AUTHOR : 'handling.team.automation@siemens.com'
FAMILY : LKinCtrl
VERSION : 5.0
//Add two coordinates (X, Y, Z) of "LKinCtrl_typeCOff3DPoint"
   VAR_INPUT 
      vIn1 : "LKinCtrl_typeCOff3DPoint";   // Input vector 1
      vIn2 : "LKinCtrl_typeCOff3DPoint";   // Input vector 2
   END_VAR


BEGIN
	//=============================================================================
	// SIEMENS AG
	// (c)Copyright 2018 All Rights Reserved
	//-----------------------------------------------------------------------------
	// Library: - 
	// Tested with: S7-1516T-3 PN
	// Engineering: TIA Portal V15
	// Restrictions: -
	// Requirements: S7-1500/S7-1500T FW 2.5
	// Functionality: Add two coordinates (X, Y, Z) of "LKinCtrl_typeCOff3DPoint"
	//-----------------------------------------------------------------------------
	// Change log table:
	// Version  Date       Expert in charge Changes applied
	// 01.00.00 2018-10-26 AW               created
	//=============================================================================
	#LKinCtrl_VecAdd.x := #vIn1.x + #vIn2.x;
	#LKinCtrl_VecAdd.y := #vIn1.y + #vIn2.y;
	#LKinCtrl_VecAdd.z := #vIn1.z + #vIn2.z;
END_FUNCTION

FUNCTION "LKinCtrl_VecAbs" : LReal
TITLE = LKinCtrl_VecAbs
{ S7_Optimized_Access := 'TRUE' }
AUTHOR : 'handling.team.automation@siemens.com'
FAMILY : LKinCtrl
VERSION : 5.0
//Calculate length of vector of coordinates (X, Y, Z) of "LKinCtrl_typeCOff3DPoint"
   VAR_INPUT 
      vIn : "LKinCtrl_typeCOff3DPoint";   // Input vector
   END_VAR


BEGIN
	//=============================================================================
	// SIEMENS AG
	// (c)Copyright 2018 All Rights Reserved
	//-----------------------------------------------------------------------------
	// Library: - 
	// Tested with: S7-1516T-3 PN
	// Engineering: TIA Portal V15
	// Restrictions: -
	// Requirements: S7-1500/S7-1500T FW 2.5
	// Functionality: Calculate length of vector of coordinates (X, Y, Z) of "LKinCtrl_typeCOff3DPoint"
	//-----------------------------------------------------------------------------
	// Change log table:
	// Version  Date       Expert in charge Changes applied
	// 01.00.00 2018-10-26 AW               created
	//=============================================================================
	
	#LKinCtrl_VecAbs := SQRT(#vIn.x * #vIn.x + #vIn.y * #vIn.y + #vIn.z * #vIn.z);
END_FUNCTION

FUNCTION "LKinCtrl_VecSub" : "LKinCtrl_typeCOff3DPoint"
TITLE = LKinCtrl_VecSub
{ S7_Optimized_Access := 'TRUE' }
AUTHOR : 'handling.team.automation@siemens.com'
FAMILY : LKinCtrl
VERSION : 5.0
//Substract two coordinates (X, Y, Z) of "LKinCtrl_typeCOff3DPoint"
   VAR_INPUT 
      vIn1 : "LKinCtrl_typeCOff3DPoint";   // Input vector 1
      vIn2 : "LKinCtrl_typeCOff3DPoint";   // Input vector 2
   END_VAR


BEGIN
	//=============================================================================
	// SIEMENS AG
	// (c)Copyright 2018 All Rights Reserved
	//-----------------------------------------------------------------------------
	// Library: - 
	// Tested with: S7-1516T-3 PN
	// Engineering: TIA Portal V15
	// Restrictions: -
	// Requirements: S7-1500/S7-1500T FW 2.5
	// Functionality: Substract two coordinates (X, Y, Z) of "LKinCtrl_typeCOff3DPoint"
	//-----------------------------------------------------------------------------
	// Change log table:
	// Version  Date       Expert in charge Changes applied
	// 01.00.00 2018-10-26 AW               created
	//=============================================================================
	#LKinCtrl_VecSub.x := #vIn1.x - #vIn2.x;
	#LKinCtrl_VecSub.y := #vIn1.y - #vIn2.y;
	#LKinCtrl_VecSub.z := #vIn1.z - #vIn2.z;
	
	
END_FUNCTION

FUNCTION "LKinCtrl_CalcVecDistancePathPlane" : Word
TITLE = LKinCtrl_CalcVecDistancePathPlane
{ S7_Optimized_Access := 'TRUE' }
AUTHOR : 'handling.team.automation@siemens.com'
FAMILY : LKinCtrl
VERSION : 5.0
//Calculate vector distance with respect to path plane
   VAR_INPUT 
      vectorInA : "LKinCtrl_typeCOff3DPoint";   // Vector A
      vectorInB : "LKinCtrl_typeCOff3DPoint";   // vector B
      pathPlane : Int;   // Path plane: XZ= 0, YZ=1, XY= 2
   END_VAR

   VAR_OUTPUT 
      distancePathPlane : LReal;   // Distance with respect to path plane
   END_VAR

   VAR_TEMP 
      tempVectorA : "LKinCtrl_typeCOff3DPoint";
      tempVectorB : "LKinCtrl_typeCOff3DPoint";
   END_VAR

   VAR CONSTANT 
      ERR_COFF_INVALID_PATH_PLANE : Word := 16#8303;   // Error - invalid path plane
   END_VAR


BEGIN
	//=============================================================================
	// SIEMENS AG
	// (c)Copyright 2019 All Rights Reserved
	//-----------------------------------------------------------------------------
	// Library: - 
	// Tested with: S7-1516T-3 PN
	// Engineering: TIA Portal V15
	// Restrictions: -
	// Requirements: S7-1500/S7-1500T FW 2.5
	// Functionality: Calculate vector distance with respect to path plane
	//-----------------------------------------------------------------------------
	// Change log table:
	// Version  Date       Expert in charge Changes applied
	// 01.00.00 2019-02-15 AW               created
	//=============================================================================
	REGION PLAUSIBILITY_CHECK
	  // Check path plane
	  IF ((#pathPlane >= "CP_XZ") AND (#pathPlane <= "CP_XY"))
	  THEN
	    ;
	  ELSE
	    #LKinCtrl_CalcVecDistancePathPlane := #ERR_COFF_INVALID_PATH_PLANE; // Invalid path plane
	    RETURN;
	  END_IF;
	END_REGION PLAUSIBILITY_CHECK
	
	
	REGION CALCULATION
	  #tempVectorA := #vectorInA;
	  #tempVectorB := #vectorInB;
	  
	  // Eleminate "third" coordinate
	  CASE #pathPlane OF
	    "CP_XY":
	      #tempVectorA.z := 0.0;
	      #tempVectorB.z := 0.0;
	      
	    "CP_XZ":
	      #tempVectorA.y := 0.0;
	      #tempVectorB.y := 0.0;
	      
	    "CP_YZ":
	      #tempVectorA.x := 0.0;
	      #tempVectorB.x := 0.0;
	  END_CASE;
	
	  #distancePathPlane := "LKinCtrl_VecAbs"("LKinCtrl_VecSub"(vIn1:=#tempVectorB, vIn2:=#tempVectorA));
	  
	  
	  
	END_REGION CALCULATION
	
	#LKinCtrl_CalcVecDistancePathPlane := 0; // o.k.
END_FUNCTION

FUNCTION "LKinCtrl_CalcCircEndPointWithGivenCenterAndAngle" : Word
TITLE = LKinCtrl_CalcCircEndPointWithGivenCenterAndAngle
{ S7_Optimized_Access := 'TRUE' }
AUTHOR : 'handling.team.automation@siemens.com'
FAMILY : LKinCtrl
VERSION : 5.0
//Calculate circle end point with given start point, circle center and angle
   VAR_INPUT 
      circleStartPoint : "LKinCtrl_typeCOff3DPoint";   // Circle start point
      circleCenterPoint : "LKinCtrl_typeCOff3DPoint";   // Circle center point
      pathPlane : Int;   // Path plane: XZ= 0, YZ=1, XY= 2
      pathChoice : DInt;   // Circle path choice: positive= 0, negative= 1
      angle : LReal;   // Circle angle
   END_VAR

   VAR_OUTPUT 
      endPoint : "LKinCtrl_typeCOff3DPoint";
   END_VAR

   VAR_TEMP 
      tempSin : LReal;
      tempCos : LReal;
      tempVOrthogonal : "LKinCtrl_typeCOff3DPoint";   // Othogonal vector
      tempVRotated : "LKinCtrl_typeCOff3DPoint";
   END_VAR

   VAR CONSTANT 
      ERR_COFF_INVALID_PATH_PLANE : Word := 16#8303;   // Error - invalid path plane
      ERR_COFF_INVALID_COMPENSATION_DIRECTION : Word := 16#8304;   // Error - invalid compensation direction
   END_VAR


BEGIN
	//=============================================================================
	// SIEMENS AG
	// (c)Copyright 2019 All Rights Reserved
	//-----------------------------------------------------------------------------
	// Library: - 
	// Tested with: S7-1516T-3 PN
	// Engineering: TIA Portal V15
	// Restrictions: -
	// Requirements: S7-1500/S7-1500T FW 2.5
	// Functionality: Calculate circle end point with given
	// start point, circle center and angle
	//-----------------------------------------------------------------------------
	// Change log table:
	// Version  Date       Expert in charge Changes applied
	// 01.00.00 2019-01-24 AW               created
	//=============================================================================
	
	REGION PLAUSIBILITY_CHECK
	  // Check path plane
	  IF ((#pathPlane >= "CP_XZ") AND (#pathPlane <= "CP_XY"))
	  THEN
	    // Check compensation direction
	    IF ((#pathChoice >= 0) AND (#pathChoice <= 1))
	    THEN
	      ;
	    ELSE
	      #LKinCtrl_CalcCircEndPointWithGivenCenterAndAngle := #ERR_COFF_INVALID_COMPENSATION_DIRECTION; // Invalid compensation direction
	      RETURN;
	    END_IF;
	  ELSE
	    #LKinCtrl_CalcCircEndPointWithGivenCenterAndAngle := #ERR_COFF_INVALID_PATH_PLANE; // Invalid path plane
	    RETURN;
	  END_IF;
	END_REGION PLAUSIBILITY_CHECK
	
	REGION CALCULATION
	  
	// Calc radius vector (difference vector) circle center to start point
	#tempVOrthogonal := "LKinCtrl_VecSub"(vIn1 := #circleStartPoint, vIn2 := #circleCenterPoint);
	
	IF (#pathChoice = 0) THEN
	  // positive
	  #tempSin := SIN(#angle * "LKINCTRL_PI" / 180.0);
	  #tempCos := COS(#angle * "LKINCTRL_PI" / 180.0);
	ELSE
	  #tempSin := SIN(- #angle * "LKINCTRL_PI" / 180.0);
	  #tempCos := COS(- #angle * "LKINCTRL_PI" / 180.0);
	END_IF;
	
	// Check path plane
	IF (#pathPlane = "CP_XY") THEN
	  // Rotation around Z
	  #tempVRotated.x := #tempVOrthogonal.x * #tempCos - #tempVOrthogonal.y * #tempSin;      // Calculation X
	  #tempVRotated.y := #tempVOrthogonal.x * #tempSin + #tempVOrthogonal.y * #tempCos;      // Calculation Y
	  #tempVRotated.z := #tempVOrthogonal.z;                                                 // Calculation Z
	  
	ELSIF (#pathPlane = "CP_XZ") THEN
	  // Rotation around Y
	  #tempVRotated.x := #tempVOrthogonal.x * #tempCos + #tempVOrthogonal.z * #tempSin;      // Calculation X
	  #tempVRotated.y := #tempVOrthogonal.y;                                                 // Calculation Y
	  #tempVRotated.z := -#tempVOrthogonal.x * #tempSin + #tempVOrthogonal.z * #tempCos;     // Calculation Z
	  
	ELSIF (#pathPlane = "CP_YZ") THEN
	  // Rotation around X
	  #tempVRotated.x := #tempVOrthogonal.x;      // Calculation X
	  #tempVRotated.y := #tempVOrthogonal.y * #tempCos - #tempVOrthogonal.z * #tempSin;       // Calculation Y
	  #tempVRotated.z := #tempVOrthogonal.y * #tempSin + #tempVOrthogonal.z * #tempCos;     // Calculation Z
	END_IF;
	
	// Calculate end point of circle by adding the rotated vector to the circle center point
	#endPoint := "LKinCtrl_VecAdd"(vIn1:=#tempVRotated, vIn2:=#circleCenterPoint);
	
	END_REGION CALCULATION
	
	#LKinCtrl_CalcCircEndPointWithGivenCenterAndAngle := 0;
END_FUNCTION

FUNCTION "LKinCtrl_CalcLineTangOrthPathPlane" : Word
TITLE = LKinCtrl_CalcLineTangOrthPathPlane
{ S7_Optimized_Access := 'TRUE' }
AUTHOR : 'handling.team.automation@siemens.com'
FAMILY : LKinCtrl
VERSION : 5.0
//Calculate orthogonal and tangential vector of a line with respect ot the path plane
   VAR_INPUT 
      pathPlane : Int;   // Path plane: XZ= 0, YZ=1, XY= 2
      compDirection : Int;   // Tool radius compensation direction: left=1, right = 0
      vInFirst : "LKinCtrl_typeCOff3DPoint";   // Next position
      vInSecond : "LKinCtrl_typeCOff3DPoint";   // Current position
   END_VAR

   VAR_OUTPUT 
      vUnitTangentialPathPlane : "LKinCtrl_typeCOff3DPoint";   // Output tangential vector - path plane - unit vector
      vUnitOrthogonalPathPlane : "LKinCtrl_typeCOff3DPoint";   // Output orthogonal vector - path plane - unit vector
   END_VAR

   VAR_TEMP 
      tempVOrthogonal : "LKinCtrl_typeCOff3DPoint";   // Othogonal vector
      tempVTangential : "LKinCtrl_typeCOff3DPoint";   // Tangential vector
   END_VAR

   VAR CONSTANT 
      ERR_COFF_INVALID_PATH_PLANE : Word := 16#8303;   // Error - invalid path plane
      ERR_COFF_INVALID_COMPENSATION_DIRECTION : Word := 16#8304;   // Error - invalid compensation direction
   END_VAR


BEGIN
	//=============================================================================
	// SIEMENS AG
	// (c)Copyright 2019 All Rights Reserved
	//-----------------------------------------------------------------------------
	// Library: - 
	// Tested with: S7-1516T-3 PN
	// Engineering: TIA Portal V15
	// Restrictions: -
	// Requirements: S7-1500/S7-1500T FW 2.5
	// Functionality: Calculate orthogonal and tangential vector of a line
	// with respect ot the path plane
	//-----------------------------------------------------------------------------
	// Change log table:
	// Version  Date       Expert in charge Changes applied
	// 01.00.00 2019-02-05 AW               created
	//=============================================================================
	
	REGION PLAUSIBILITY_CHECK
	// Check path plane
	  IF ((#pathPlane >= "CP_XZ") AND (#pathPlane <= "CP_XY"))
	THEN
	  // Check compensation direction
	  IF ((#compDirection >= "LKINCTRL_COMP_LEFT") AND (#compDirection <= "LKINCTRL_COMP_RIGHT"))
	  THEN
	    ;
	  ELSE
	    #LKinCtrl_CalcLineTangOrthPathPlane := #ERR_COFF_INVALID_COMPENSATION_DIRECTION; // Invalid compensation direction
	    RETURN;
	  END_IF;
	ELSE
	  #LKinCtrl_CalcLineTangOrthPathPlane := #ERR_COFF_INVALID_PATH_PLANE; // Invalid path plane
	  RETURN;
	END_IF;
	
	END_REGION PLAUSIBILITY_CHECK
	
	REGION CALCULATION
	  // Calculate difference vector (take care of path plane) - tangential vector
	  #tempVTangential := "LKinCtrl_VecSub"(vIn1 := #vInFirst,
	                                        vIn2 := #vInSecond);
	  
	  // Take care of path plane
	  CASE #pathPlane OF
	    "CP_XY":
	      #tempVTangential.z := 0.0;
	      
	    "CP_XZ":
	      #tempVTangential.y := 0.0;
	      
	    "CP_YZ":
	      #tempVTangential.x := 0.0;
	  END_CASE;
	  
	  // Normalize vector
	  #tempVTangential := "LKinCtrl_VecUnit"(vIn := #tempVTangential);
	  
	  
	// Calculate orthogonal vector to current vector depending on path plane and compensation direction
	CASE #pathPlane OF
	  "CP_XY":
	    IF (#compDirection = "LKINCTRL_COMP_LEFT") THEN
	      #tempVOrthogonal.x := - #tempVTangential.y;
	      #tempVOrthogonal.y := #tempVTangential.x;
	      #tempVOrthogonal.z := 0.0;
	    ELSE
	      #tempVOrthogonal.x := #tempVTangential.y;
	      #tempVOrthogonal.y := - #tempVTangential.x;
	      #tempVOrthogonal.z := 0.0;          
	    END_IF;
	    
	  "CP_XZ":
	    (*
	    IF (#compDirection = "LKINCTRL_COMP_LEFT") THEN
	      #tempVOrthogonal.x := #tempVTangential.z;
	      #tempVOrthogonal.y := 0.0;
	      #tempVOrthogonal.z := - #tempVTangential.x;
	    ELSE
	      #tempVOrthogonal.x := - #tempVTangential.z;
	      #tempVOrthogonal.y := 0.0;
	      #tempVOrthogonal.z := #tempVTangential.x;
	    END_IF;*)
	    
	    IF (#compDirection = "LKINCTRL_COMP_LEFT") THEN
	      #tempVOrthogonal.x := -#tempVTangential.z;
	      #tempVOrthogonal.y := 0.0;
	      #tempVOrthogonal.z := #tempVTangential.x;
	    ELSE
	      #tempVOrthogonal.x := #tempVTangential.z;
	      #tempVOrthogonal.y := 0.0;
	      #tempVOrthogonal.z := -#tempVTangential.x;
	    END_IF;
	    
	  "CP_YZ":
	    IF (#compDirection = "LKINCTRL_COMP_LEFT") THEN
	      #tempVOrthogonal.x := 0.0;
	      #tempVOrthogonal.y := - #tempVTangential.z;
	      #tempVOrthogonal.z := #tempVTangential.y;
	    ELSE
	      #tempVOrthogonal.x := 0.0;
	      #tempVOrthogonal.y := #tempVTangential.z;
	      #tempVOrthogonal.z := - #tempVTangential.y;
	    END_IF;
	END_CASE;
	END_REGION CALCULATION
	
	#vUnitTangentialPathPlane := #tempVTangential;
	#vUnitOrthogonalPathPlane := #tempVOrthogonal;
	#LKinCtrl_CalcLineTangOrthPathPlane := 0;
	
	
	
END_FUNCTION

FUNCTION "LKinCtrl_VecUnit" : "LKinCtrl_typeCOff3DPoint"
TITLE = LKinCtrl_VecUnit
{ S7_Optimized_Access := 'TRUE' }
AUTHOR : 'handling.team.automation@siemens.com'
FAMILY : LKinCtrl
VERSION : 5.0
//Create unit vector of coordinates (X, Y, Z) of "LKinCtrl_typeCOff3DPoint"
   VAR_INPUT 
      vIn : "LKinCtrl_typeCOff3DPoint";   // Input vector
   END_VAR


BEGIN
	//=============================================================================
	// SIEMENS AG
	// (c)Copyright 2018 All Rights Reserved
	//-----------------------------------------------------------------------------
	// Library: - 
	// Tested with: S7-1516T-3 PN
	// Engineering: TIA Portal V15
	// Restrictions: -
	// Requirements: S7-1500/S7-1500T FW 2.5
	// Functionality: Create unit vector of coordinates (X, Y, Z) of "LKinCtrl_typeCOff3DPoint"
	//-----------------------------------------------------------------------------
	// Change log table:
	// Version  Date       Expert in charge Changes applied
	// 01.00.00 2018-08-27 SF               created
	//=============================================================================
	
	//Out = In/abs(In)
	#LKinCtrl_VecUnit := "LKinCtrl_VecDivScal"(vIn := #vIn,
	                                           sIn := "LKinCtrl_VecAbs"(#vIn));
	
	
END_FUNCTION

FUNCTION "LKinCtrl_VecDivScal" : "LKinCtrl_typeCOff3DPoint"
TITLE = LKinCtrl_VecDivScal
{ S7_Optimized_Access := 'TRUE' }
AUTHOR : 'handling.team.automation@siemens.com'
FAMILY : LKinCtrl
VERSION : 5.0
//Divide coordinate with scalar of coordinates (X, Y, Z) of "LKinCtrl_typeCOff3DPoint"
   VAR_INPUT 
      vIn : "LKinCtrl_typeCOff3DPoint";   // Input vector
      sIn : LReal;   // Input scalar
   END_VAR


BEGIN
	//=============================================================================
	// SIEMENS AG
	// (c)Copyright 2018 All Rights Reserved
	//-----------------------------------------------------------------------------
	// Library: - 
	// Tested with: S7-1516T-3 PN
	// Engineering: TIA Portal V15
	// Restrictions: -
	// Requirements: S7-1500/S7-1500T FW 2.5
	// Functionality: Divide coordinate with scalar of coordinates (X, Y, Z) of "LKinCtrl_typeCOff3DPoint"
	//-----------------------------------------------------------------------------
	// Change log table:
	// Version  Date       Expert in charge Changes applied
	// 01.00.00 2018-10-26 AW               created
	//=============================================================================
	
	IF (#sIn <> 0.0) THEN
	  #LKinCtrl_VecDivScal.x := #vIn.x / #sIn;
	  #LKinCtrl_VecDivScal.y := #vIn.y / #sIn;
	  #LKinCtrl_VecDivScal.z := #vIn.z / #sIn;
	ELSE
	  #LKinCtrl_VecDivScal.x := 0.0;
	  #LKinCtrl_VecDivScal.y := 0.0;
	  #LKinCtrl_VecDivScal.z := 0.0;
	END_IF;
END_FUNCTION

FUNCTION "LKinCtrl_VecScale" : "LKinCtrl_typeCOff3DPoint"
TITLE = LKinCtrl_VecScale
{ S7_Optimized_Access := 'TRUE' }
AUTHOR : 'handling.team.automation@siemens.com'
FAMILY : LKinCtrl
VERSION : 5.0
//Scale vector (X, Y, Z) of "LKinCtrl_typeCOff3DPoint"
   VAR_INPUT 
      vIn : "LKinCtrl_typeCOff3DPoint";   // Input vector
      factor : LReal;   // Scaling factor
   END_VAR


BEGIN
	//=============================================================================
	// SIEMENS AG
	// (c)Copyright 2018 All Rights Reserved
	//-----------------------------------------------------------------------------
	// Library: - 
	// Tested with: S7-1516T-3 PN
	// Engineering: TIA Portal V15
	// Restrictions: -
	// Requirements: S7-1500/S7-1500T FW 2.5
	// Functionality: Scale vector (X, Y, Z) of "LKinCtrl_typeCOff3DPoint"
	//-----------------------------------------------------------------------------
	// Change log table:
	// Version  Date       Expert in charge Changes applied
	// 01.00.00 2018-10-26 AW               created
	//=============================================================================
	
	#LKinCtrl_VecScale.x := #vIn.x * #factor;
	#LKinCtrl_VecScale.y := #vIn.y * #factor;
	#LKinCtrl_VecScale.z := #vIn.z * #factor;
	
END_FUNCTION

FUNCTION "LKinCtrl_CalcLineLineIntersectionPoint" : Word
TITLE = LKinCtrl_CalcLineLineIntersectionPoint
{ S7_Optimized_Access := 'TRUE' }
AUTHOR : 'handling.team.automation@siemens.com'
FAMILY : LKinCtrl
VERSION : 5.0
//Calculate the line segment Pa/Pb that is the shortest route between two lines P1P2 and P3P4
   VAR_INPUT 
      startPointFirstLine : "LKinCtrl_typeCOff3DPoint";   // Start point first line
      endPointFirstLine : "LKinCtrl_typeCOff3DPoint";   // End point first line
      startPointSecondLine : "LKinCtrl_typeCOff3DPoint";   // Start point second line
      endPointSecondLine : "LKinCtrl_typeCOff3DPoint";   // End point second line
   END_VAR

   VAR_OUTPUT 
      intersectionPointA : "LKinCtrl_typeCOff3DPoint";   // Intersection point a
      intersectionPointB : "LKinCtrl_typeCOff3DPoint";   // Intersection point b
      muA : LReal;   // Direction vector a
      muB : LReal;   // Direction vector b
   END_VAR

   VAR_TEMP 
      tempP13 : "LKinCtrl_typeCOff3DPoint";
      tempP43 : "LKinCtrl_typeCOff3DPoint";
      tempP21 : "LKinCtrl_typeCOff3DPoint";
      tempD1343 : LReal;
      tempD4321 : LReal;
      tempD1321 : LReal;
      tempD4343 : LReal;
      tempD2121 : LReal;
      tempNumer : LReal;
      tempDenom : LReal;
   END_VAR

   VAR CONSTANT 
      COFF_EPS : LReal := 0.001;   // Internal constant
      ERR_COFF_LINES_DO_NOT_INTERSECT : Word := 16#8312;   // Error - no solution, lines don't intersect
      ERR_COFF_ZERO_VECTOR : Word := 16#8313;   // Error - zero vector
   END_VAR


BEGIN
	//=============================================================================
	// SIEMENS AG
	// (c)Copyright 2019 All Rights Reserved
	//-----------------------------------------------------------------------------
	// Library: - 
	// Tested with: S7-1516T-3 PN
	// Engineering: TIA Portal V15
	// Restrictions: -
	// Requirements: S7-1500/S7-1500T FW 2.5
	// Functionality: Calculate the line segment Pa/Pb that is the shortest route
	// between two lines P1P2 and P3P4. Calculate also the values of mua and mub where
	// Pa = P1 + mua (P2 - P1)
	// Pb = P3 + mub (P4 - P3)
	// Return error if the lines don't intersect
	//-----------------------------------------------------------------------------
	// Change log table:
	// Version  Date       Expert in charge Changes applied
	// 01.00.00 2019-02-05 AW               created
	//=============================================================================
	REGION PLAUSIBILITY_CHECK
	
	END_REGION PLAUSIBILITY_CHECK
	
	REGION CALCULATION
	  #tempP13.x := #startPointFirstLine.x - #startPointSecondLine.x;
	  #tempP13.y := #startPointFirstLine.y - #startPointSecondLine.y;
	  #tempP13.z := #startPointFirstLine.z - #startPointSecondLine.z;
	  #tempP43.x := #endPointSecondLine.x - #startPointSecondLine.x;
	  #tempP43.y := #endPointSecondLine.y - #startPointSecondLine.y;
	  #tempP43.z := #endPointSecondLine.z - #startPointSecondLine.z;
	  IF ((ABS(#tempP43.x) < #COFF_EPS) AND (ABS(#tempP43.y) < #COFF_EPS) AND (ABS(#tempP43.z) < #COFF_EPS)) THEN
	    #LKinCtrl_CalcLineLineIntersectionPoint := #ERR_COFF_LINES_DO_NOT_INTERSECT;
	    RETURN;
	  END_IF;
	  
	  #tempP21.x := #endPointFirstLine.x - #startPointFirstLine.x;
	  #tempP21.y := #endPointFirstLine.y - #startPointFirstLine.y;
	  #tempP21.z := #endPointFirstLine.z - #startPointFirstLine.z;
	  IF ((ABS(#tempP21.x) < #COFF_EPS) AND (ABS(#tempP21.y) < #COFF_EPS) AND (ABS(#tempP21.z) < #COFF_EPS)) THEN
	    #LKinCtrl_CalcLineLineIntersectionPoint := #ERR_COFF_LINES_DO_NOT_INTERSECT;
	    RETURN;
	  END_IF;
	  
	  #tempD1343 := #tempP13.x * #tempP43.x + #tempP13.y * #tempP43.y + #tempP13.z * #tempP43.z;
	  #tempD4321 := #tempP43.x * #tempP21.x + #tempP43.y * #tempP21.y + #tempP43.z * #tempP21.z;
	  #tempD1321 := #tempP13.x * #tempP21.x + #tempP13.y * #tempP21.y + #tempP13.z * #tempP21.z;
	  #tempD4343 := #tempP43.x * #tempP43.x + #tempP43.y * #tempP43.y + #tempP43.z * #tempP43.z;
	  #tempD2121 := #tempP21.x * #tempP21.x + #tempP21.y * #tempP21.y + #tempP21.z * #tempP21.z;
	  
	  #tempDenom := #tempD2121 * #tempD4343 - #tempD4321 * #tempD4321;
	  IF (ABS(#tempDenom) < #COFF_EPS) THEN
	    #LKinCtrl_CalcLineLineIntersectionPoint := #ERR_COFF_LINES_DO_NOT_INTERSECT;
	    RETURN;
	  END_IF;
	  
	  #tempNumer := #tempD1343 * #tempD4321 - #tempD1321 * #tempD4343;
	  
	  #muA := #tempNumer / #tempDenom;
	  #muB := (#tempD1343 + #tempD4321 * #muA) / #tempD4343;
	  
	  #intersectionPointA.x := #startPointFirstLine.x + #muA * #tempP21.x;
	  #intersectionPointA.y := #startPointFirstLine.y + #muA * #tempP21.y;
	  #intersectionPointA.z := #startPointFirstLine.z + #muA * #tempP21.z;
	
	  #intersectionPointB.x := #startPointSecondLine.x + #muB * #tempP43.x;
	  #intersectionPointB.y := #startPointSecondLine.y + #muB * #tempP43.y;
	  #intersectionPointB.z := #startPointSecondLine.z + #muB * #tempP43.z;
	  
	END_REGION
	#LKinCtrl_CalcLineLineIntersectionPoint := 0;
END_FUNCTION

FUNCTION "LKinCtrl_CheckInnerOuterCorner" : Word
TITLE = LKinCtrl_CheckInnerOuterCorner
{ S7_Optimized_Access := 'TRUE' }
AUTHOR : 'handling.team.automation@siemens.com'
FAMILY : LKinCtrl
VERSION : 5.0
//Check for inner or outer corner
   VAR_INPUT 
      vInFirst : "LKinCtrl_typeCOff3DPoint";   // Input vector first
      vInSecond : "LKinCtrl_typeCOff3DPoint";   // Input vector second
      pathPlane : Int;   // Path plane: XZ= 0, YZ=1, XY= 2
      direction : Int;   // Tool radius compensation direction: left=1, right = 0
   END_VAR

   VAR_OUTPUT 
      cornerType : Int;   // Corner type - 0: outer corner, 1: inner corner
   END_VAR

   VAR_TEMP 
      tempCrossVec : "LKinCtrl_typeCOff3DPoint";
   END_VAR

   VAR CONSTANT 
      ERR_COFF_INVALID_PATH_PLANE : Word := 16#8303;   // Invalid path plane
      ERR_COFF_INVALID_COMPENSATION_DIRECTION : Word := 16#8304;   // Invalid compensation direction
   END_VAR


BEGIN
	//=============================================================================
	// SIEMENS AG
	// (c)Copyright 2019 All Rights Reserved
	//-----------------------------------------------------------------------------
	// Library: - 
	// Tested with: S7-1516T-3 PN
	// Engineering: TIA Portal V15
	// Restrictions: -
	// Requirements: S7-1500/S7-1500T FW 2.5
	// Functionality: Check for inner or outer corner
	//-----------------------------------------------------------------------------
	// Change log table:
	// Version  Date       Expert in charge Changes applied
	// 01.00.00 2019-01-24 AW               created
	// 01.00.01 2020-10-13 AW               bugfix - path plane CP_XZ - different orientation, not against third axis!
	//=============================================================================
	REGION PLAUSIBILITY_CHECK
	  // Check path plane
	  IF ((#pathPlane >= "CP_XZ") AND (#pathPlane <= "CP_XY"))
	  THEN
	    // Check compensation direction
	    IF ((#direction >= "LKINCTRL_COMP_LEFT") AND (#direction <= "LKINCTRL_COMP_RIGHT"))
	    THEN
	      ;
	    ELSE
	      #LKinCtrl_CheckInnerOuterCorner := #ERR_COFF_INVALID_COMPENSATION_DIRECTION; // Invalid compensation direction
	      RETURN;
	    END_IF;
	  ELSE
	    #LKinCtrl_CheckInnerOuterCorner := #ERR_COFF_INVALID_PATH_PLANE; // Invalid path plane
	    RETURN;
	  END_IF;
	END_REGION PLAUSIBILITY_CHECK
	
	REGION CALCULATION
	  #tempCrossVec := "LKinCtrl_VecCrossProd"(vIn1 := #vInFirst,
	                                           vIn2 := #vInSecond);
	  
	// Check path plane
	IF (#pathPlane = "CP_XY") THEN
	  IF (#direction = "LKINCTRL_COMP_RIGHT") THEN
	    IF (#tempCrossVec.z > 0.0) THEN
	      #cornerType := "LKINCTRL_OUTER_CORNER";
	    ELSE
	      #cornerType := "LKINCTRL_INNER_CORNER";
	    END_IF;
	  ELSE
	    IF (#tempCrossVec.z < 0.0) THEN
	      #cornerType := "LKINCTRL_OUTER_CORNER";
	    ELSE
	      #cornerType := "LKINCTRL_INNER_CORNER";
	    END_IF;
	  END_IF;
	  
	// 2020-10-13 AW path plane CP_XZ - different orientation, not against third axis!
	// direction changed
	ELSIF (#pathPlane = "CP_XZ") THEN
	    IF (#direction = "LKINCTRL_COMP_RIGHT") THEN
	      IF (#tempCrossVec.y > 0.0) THEN
	        #cornerType := "LKINCTRL_INNER_CORNER";
	      ELSE
	        #cornerType := "LKINCTRL_OUTER_CORNER";
	      END_IF;
	    ELSE
	      IF (#tempCrossVec.y < 0.0) THEN
	        #cornerType := "LKINCTRL_INNER_CORNER";
	      ELSE
	        #cornerType := "LKINCTRL_OUTER_CORNER";
	      END_IF;
	    END_IF;
	  ELSIF (#pathPlane = "CP_YZ") THEN
	  IF (#direction = "LKINCTRL_COMP_RIGHT") THEN
	    IF (#tempCrossVec.x > 0.0) THEN
	      #cornerType := "LKINCTRL_OUTER_CORNER";
	    ELSE
	      #cornerType := "LKINCTRL_INNER_CORNER";
	    END_IF;
	  ELSE
	    IF (#tempCrossVec.x < 0.0) THEN
	      #cornerType := "LKINCTRL_OUTER_CORNER";
	    ELSE
	      #cornerType := "LKINCTRL_INNER_CORNER";
	    END_IF;
	  END_IF;
	END_IF;
	
	#LKinCtrl_CheckInnerOuterCorner := 0;
	END_REGION CALCULATION
END_FUNCTION

FUNCTION "LKinCtrl_VecCrossProd" : "LKinCtrl_typeCOff3DPoint"
TITLE = LKinCtrl_VecCrossProd
{ S7_Optimized_Access := 'TRUE' }
AUTHOR : 'handling.team.automation@siemens.com'
FAMILY : LKinCtrl
VERSION : 5.0
//Cross product of two coordinates (X, Y, Z) of "LKinCtrl_typeCOff3DPoint"
   VAR_INPUT 
      vIn1 : "LKinCtrl_typeCOff3DPoint";   // Input vector 1
      vIn2 : "LKinCtrl_typeCOff3DPoint";   // Input vector 2
   END_VAR


BEGIN
	//=============================================================================
	// SIEMENS AG
	// (c)Copyright 2018 All Rights Reserved
	//-----------------------------------------------------------------------------
	// Library: - 
	// Tested with: S7-1516T-3 PN
	// Engineering: TIA Portal V15
	// Restrictions: -
	// Requirements: S7-1500/S7-1500T FW 2.5
	// Functionality: Cross product of two coordinates (X, Y, Z) of "LKinCtrl_typeCOff3DPoint"
	//-----------------------------------------------------------------------------
	// Change log table:
	// Version  Date       Expert in charge Changes applied
	// 01.00.00 2019-01-24 AW               created
	//=============================================================================
	
	#LKinCtrl_VecCrossProd.x := #vIn1.y * #vIn2.z - #vIn1.z * #vIn2.y;
	#LKinCtrl_VecCrossProd.y := #vIn1.z * #vIn2.x - #vIn1.x * #vIn2.z;
	#LKinCtrl_VecCrossProd.z := #vIn1.x * #vIn2.y - #vIn1.y * #vIn2.x;
	
	
END_FUNCTION

FUNCTION "LKinCtrl_CalcCircleIntermediatePos" : Void
TITLE = LKinCtrl_CalcCircleIntermediatePos
{ S7_Optimized_Access := 'TRUE' }
AUTHOR : 'handling.team.automation@siemens.com'
FAMILY : LKinCtrl
VERSION : 5.0
//Calculate intermediate point of circle with given initial end point, calculated end point and tool radius
   VAR_INPUT 
      initialEndPoint : "LKinCtrl_typeCOff3DPoint";   // Initial end point
      newEndPoint : "LKinCtrl_typeCOff3DPoint";   // New calculated end point
      toolRadius : LReal;   // Tool radius
   END_VAR

   VAR_OUTPUT 
      circIntermediatePoint : "LKinCtrl_typeCOff3DPoint";   // circle intermediate point
   END_VAR

   VAR_TEMP 
      tempVecDiff : "LKinCtrl_typeCOff3DPoint";
      tempUnitVecDiff : "LKinCtrl_typeCOff3DPoint";
   END_VAR


BEGIN
	//=============================================================================
	// SIEMENS AG
	// (c)Copyright 2019 All Rights Reserved
	//-----------------------------------------------------------------------------
	// Library: - 
	// Tested with: S7-1516T-3 PN
	// Engineering: TIA Portal V15
	// Restrictions: -
	// Requirements: S7-1500/S7-1500T FW 2.5
	// Functionality: Calculate intermediate point of circle
	// with given initial end point, calculated end point and tool radius
	//-----------------------------------------------------------------------------
	// Change log table:
	// Version  Date       Expert in charge Changes applied
	// 01.00.00 2019-02-05 AW               created
	//=============================================================================
	
	REGION PLAUSIBILITY_CHECK
	END_REGION PLAUSIBILITY_CHECK
	
	REGION CALCULATION
	// Difference vector between new end point and initial end point
	#tempVecDiff := "LKinCtrl_VecSub"(vIn1 := #newEndPoint,
	                               vIn2 := #initialEndPoint);
	 
	// Calculate direction vetor to intermediate point
	#tempUnitVecDiff := "LKinCtrl_VecUnit"(#tempVecDiff);
	
	// Calculate intermediate point: initialEndPoint + lambda * radius
	#circIntermediatePoint := "LKinCtrl_VecAdd"(vIn1:= #initialEndPoint, vIn2:= "LKinCtrl_VecScale"(vIn := #tempUnitVecDiff, factor := #toolRadius));
	
	END_REGION CALCULATION
END_FUNCTION

FUNCTION "LKinCtrl_CalcCircCenterByIntermediatePointAndEndPoint" : Word
TITLE = LKinCtrl_CalcCircCenterByIntermediatePointAndEndPoint
{ S7_Optimized_Access := 'TRUE' }
AUTHOR : 'handling.team.automation@siemens.com'
FAMILY : LKinCtrl
VERSION : 5.0
//Calculate circle center point with given intermediate point
   VAR_INPUT 
      circleStartPoint : "LKinCtrl_typeCOff3DPoint";   // Circle start point
      circleEndPoint : "LKinCtrl_typeCOff3DPoint";   // Circle end point
      circleIntermediatePoint : "LKinCtrl_typeCOff3DPoint";   // Circle intermediate point
      pathPlane : Int;   // Path plane: XZ= 0, YZ=1, XY= 2
   END_VAR

   VAR_OUTPUT 
      circleCenterPoint : "LKinCtrl_typeCOff3DPoint";   // Circle center point
   END_VAR

   VAR_TEMP 
      tempVecL : "LKinCtrl_typeCOff3DPoint";
      tempVecP1P2 : "LKinCtrl_typeCOff3DPoint";
      tempVecP3P4 : "LKinCtrl_typeCOff3DPoint";
      tempLengthVecP1P2 : LReal;
      tempLengthVecP3P4 : LReal;
      tempUnitVecP1P2 : "LKinCtrl_typeCOff3DPoint";
      tempUnitVecP3P4 : "LKinCtrl_typeCOff3DPoint";
      tempP12 : "LKinCtrl_typeCOff3DPoint";
      tempP34 : "LKinCtrl_typeCOff3DPoint";
      tempP123 : "LKinCtrl_typeCOff3DPoint";
      tempP341 : "LKinCtrl_typeCOff3DPoint";
      tempOrthVecP1P2 : "LKinCtrl_typeCOff3DPoint";
      tempOrthVecP3P4 : "LKinCtrl_typeCOff3DPoint";
      tempRetValue : Word;
      tempPa : "LKinCtrl_typeCOff3DPoint";
      tempPb : "LKinCtrl_typeCOff3DPoint";
      tempMua : LReal;
      tempMub : LReal;
   END_VAR

   VAR CONSTANT 
      ERR_COFF_INVALID_PATH_PLANE : Word := 16#8303;   // Error - invalid path plane
   END_VAR


BEGIN
	//=============================================================================
	// SIEMENS AG
	// (c)Copyright 2019 All Rights Reserved
	//-----------------------------------------------------------------------------
	// Library: - 
	// Tested with: S7-1516T-3 PN
	// Engineering: TIA Portal V15
	// Restrictions: -
	// Requirements: S7-1500/S7-1500T FW 2.5
	// Functionality: Calculate circle center point with given intermediate point
	// and end point
	//-----------------------------------------------------------------------------
	// Change log table:
	// Version  Date       Expert in charge Changes applied
	// 01.00.00 2019-02-05 AW               created
	//=============================================================================
	
	
	REGION PLAUSIBILITY_CHECK
	// Check path plane
	  IF ((#pathPlane >= "CP_XZ") AND (#pathPlane <= "CP_XY"))
	THEN
	  ;
	ELSE
	  #LKinCtrl_CalcCircCenterByIntermediatePointAndEndPoint := #ERR_COFF_INVALID_PATH_PLANE; // Invalid path plane
	  RETURN;
	END_IF;
	END_REGION PLAUSIBILITY_CHECK
	
	REGION CALCULATION
	
	  // Intermediate point - start point
	  #tempVecP1P2 := "LKinCtrl_VecSub"(vIn1:= #circleIntermediatePoint, vIn2:= #circleStartPoint);
	  // Intermediate point - end point
	  #tempVecP3P4 := "LKinCtrl_VecSub"(vIn1 := #circleIntermediatePoint, vIn2 := #circleEndPoint);
	  
	  // Length of vectors
	  #tempLengthVecP1P2 := "LKinCtrl_VecAbs"(#tempVecP1P2);
	  #tempLengthVecP3P4 := "LKinCtrl_VecAbs"(#tempVecP3P4);
	
	  // Direction of vectors
	  #tempUnitVecP1P2 := "LKinCtrl_VecUnit"(#tempVecP1P2);
	  #tempUnitVecP3P4 := "LKinCtrl_VecUnit"(#tempVecP3P4);
	
	  // Perpendicular bisector
	  #tempP12 := "LKinCtrl_VecAdd"(vIn1:= #circleStartPoint, vIn2:= "LKinCtrl_VecScale"(vIn:= #tempUnitVecP1P2, factor:= (#tempLengthVecP1P2 / 2.0)));
	  #tempP34 := "LKinCtrl_VecAdd"(vIn1:= #circleEndPoint, vIn2:="LKinCtrl_VecScale"(vIn:= #tempUnitVecP3P4, factor:=(#tempLengthVecP3P4 / 2.0)));
	  
	  // Rotate vector according to path plane
	  // Calc complete shift
	  CASE #pathPlane OF
	    "CP_XY":
	        // Orthogonal end point - intermediate point
	        #tempOrthVecP1P2.x := - #tempUnitVecP1P2.y;
	        #tempOrthVecP1P2.y := #tempUnitVecP1P2.x;
	        #tempOrthVecP1P2.z := 0.0;
	        
	        // Orthogonal end point - intermediate point
	        #tempOrthVecP3P4.x := #tempUnitVecP3P4.y;
	        #tempOrthVecP3P4.y := - #tempUnitVecP3P4.x;
	        #tempOrthVecP3P4.z := 0.0;
	        
	      "CP_XZ":
	        // Orthogonal end point - intermediate point
	        #tempOrthVecP1P2.x := #tempUnitVecP1P2.z;
	        #tempOrthVecP1P2.y := 0.0;
	        #tempOrthVecP1P2.z := - #tempUnitVecP1P2.x;
	        
	        // Orthogonal end point - intermediate point
	        #tempOrthVecP3P4.x := - #tempUnitVecP3P4.z;
	        #tempOrthVecP3P4.y := 0.0;
	        #tempOrthVecP3P4.z := #tempUnitVecP3P4.x;
	        
	      "CP_YZ":
	        // Orthogonal end point - intermediate point
	        #tempOrthVecP1P2.x := 0.0;
	        #tempOrthVecP1P2.y := - #tempUnitVecP1P2.z;
	        #tempOrthVecP1P2.z := #tempUnitVecP1P2.y;
	        
	        // Orthogonal end point - intermediate point
	        #tempOrthVecP3P4.x := 0.0;
	        #tempOrthVecP3P4.y := #tempUnitVecP3P4.z;
	        #tempOrthVecP3P4.z := - #tempUnitVecP3P4.y;
	  END_CASE;
	  
	  #tempOrthVecP1P2 := "LKinCtrl_VecScale"(vIn:= #tempOrthVecP1P2, factor:= #tempLengthVecP1P2);
	  #tempOrthVecP3P4 := "LKinCtrl_VecScale"(vIn:= #tempOrthVecP3P4, factor:= #tempLengthVecP3P4);
	  
	  #tempP123 := "LKinCtrl_VecAdd"(vIn1:= #tempP12, vIn2:= #tempOrthVecP1P2);
	  #tempP341 := "LKinCtrl_VecAdd"(vIn1:= #tempP34, vIn2:= #tempOrthVecP3P4);
	  
	  #tempRetValue := "LKinCtrl_CalcLineLineIntersectionPoint"(startPointFirstLine := #tempP12,
	                                                   endPointFirstLine := #tempP123,
	                                                   startPointSecondLine := #tempP34,
	                                                   endPointSecondLine := #tempP341,
	                                                   intersectionPointA => #tempPa,
	                                                   intersectionPointB => #tempPb,
	                                                   muA => #tempMua,
	                                                   muB => #tempMub);
	  IF (#tempRetValue <> 0) THEN
	    #LKinCtrl_CalcCircCenterByIntermediatePointAndEndPoint := #tempRetValue;
	    RETURN;
	  END_IF;
	
	END_REGION CALCULATION
	
	#circleCenterPoint := #tempPa;
	
	#LKinCtrl_CalcCircCenterByIntermediatePointAndEndPoint := 0; // o.k.
END_FUNCTION

FUNCTION "LKinCtrl_CalcCircCenterByRadiusAndEndPoint" : Word
TITLE = LKinCtrl_CalcCircCenterByRadiusAndEndPoint
{ S7_Optimized_Access := 'TRUE' }
AUTHOR : 'handling.team.automation@siemens.com'
FAMILY : LKinCtrl
VERSION : 5.0
//Calculate circle center point with given start point, end point and radius
   VAR_INPUT 
      circleStartPoint : "LKinCtrl_typeCOff3DPoint";   // Circle start point
      circleEndPoint : "LKinCtrl_typeCOff3DPoint";   // Circle end point
      pathPlane : Int;   // Path plane: XZ= 0, YZ=1, XY= 2
      circleRadius : LReal;   // Circle radius
      pathChoice : DInt;   // Circle path choice: positive= 0, negative= 1
   END_VAR

   VAR_OUTPUT 
      circCenterPoint : "LKinCtrl_typeCOff3DPoint";   // Circle center point
   END_VAR

   VAR_TEMP 
      tempRetValue : Word;
      tempPa : "LKinCtrl_typeCOff3DPoint";
      tempPb : "LKinCtrl_typeCOff3DPoint";
      tempVEndStart : "LKinCtrl_typeCOff3DPoint";
      tempVPaStart : "LKinCtrl_typeCOff3DPoint";
      tempCrossVec : "LKinCtrl_typeCOff3DPoint";
   END_VAR

   VAR CONSTANT 
      ERR_COFF_INVALID_PATH_PLANE : Word := 16#8303;   // Error - invalid path plane
   END_VAR


BEGIN
	//=============================================================================
	// SIEMENS AG
	// (c)Copyright 2019 All Rights Reserved
	//-----------------------------------------------------------------------------
	// Library: - 
	// Tested with: S7-1516T-3 PN
	// Engineering: TIA Portal V15
	// Restrictions: -
	// Requirements: S7-1500/S7-1500T FW 2.5
	// Functionality: Calculate circle center point with given start point, end point and radius
	//-----------------------------------------------------------------------------
	// Change log table:
	// Version  Date       Expert in charge Changes applied
	// 01.00.00 2019-01-24 AW               created
	//=============================================================================
	
	REGION PLAUSIBILITY_CHECK
	  // Check path plane
	  IF ((#pathPlane >= "CP_XZ") AND (#pathPlane <= "CP_XY"))
	  THEN
	    ;
	  ELSE
	    #LKinCtrl_CalcCircCenterByRadiusAndEndPoint := #ERR_COFF_INVALID_PATH_PLANE; // Invalid path plane
	    RETURN;
	  END_IF;
	END_REGION PLAUSIBILITY_CHECK
	
	REGION CALCULATION
	  
	  
	  // Calculate circle center point by letting the following two circles intersect
	  // 1st circle around start point with radius
	  // 2nd circle around end point with radius
	  #tempRetValue := "LKinCtrl_CalcCircleCircleIntersectionPoint"(circleCenterPoint1 := #circleStartPoint,
	                                                                circleCenterPoint2 := #circleEndPoint,
	                                                                circleRadius1 := #circleRadius,
	                                                                circleRadius2 := #circleRadius,
	                                                                pathPlane := #pathPlane,
	                                                                intersectionPointA => #tempPa,
	                                                                intersectionPointB => #tempPb);
	
	  IF (#tempRetValue <> 16#0) THEN
	    #LKinCtrl_CalcCircCenterByRadiusAndEndPoint := #tempRetValue;
	    RETURN;
	  END_IF;
	  
	  // Which one ist the correct circle center point? Calculate left and right
	  
	  // Difference vectors
	  #tempVEndStart := "LKinCtrl_VecSub"(vIn1 := #circleEndPoint, vIn2 := #circleStartPoint);
	  #tempVPaStart := "LKinCtrl_VecSub"(vIn1 := #tempPa, vIn2 := #circleStartPoint);
	  #tempCrossVec := "LKinCtrl_VecCrossProd"(vIn1 := #tempVEndStart,
	                                           vIn2 := #tempVPaStart);
	
	  // Check path plane
	  IF (#pathPlane = "CP_XY") THEN
	    IF (#tempCrossVec.z > 0.0) THEN
	      IF (#pathChoice = 0) THEN
	        #circCenterPoint := #tempPa;
	      ELSE
	        #circCenterPoint := #tempPb;
	      END_IF;
	    ELSE
	      // Todo - is the else necessary?
	      IF (#pathChoice = 0) THEN
	        #circCenterPoint := #tempPb;
	      ELSE
	        #circCenterPoint := #tempPa;
	      END_IF;
	    END_IF;
	  ELSIF (#pathPlane = "CP_XZ") THEN
	    IF (#tempCrossVec.y > 0.0) THEN
	      IF (#pathChoice = 0) THEN
	        #circCenterPoint := #tempPa;
	      ELSE
	        #circCenterPoint := #tempPb;
	      END_IF;
	    ELSE
	      IF (#pathChoice = 0) THEN
	        #circCenterPoint := #tempPb;
	      ELSE
	        #circCenterPoint := #tempPa;
	      END_IF;
	    END_IF;
	  ELSIF (#pathPlane = "CP_YZ") THEN
	    IF (#tempCrossVec.x > 0.0) THEN
	      IF (#pathChoice = 0) THEN
	        #circCenterPoint := #tempPa;
	      ELSE
	        #circCenterPoint := #tempPb;
	      END_IF;
	    ELSE
	      IF (#pathChoice = 0) THEN
	        #circCenterPoint := #tempPb;
	      ELSE
	        #circCenterPoint := #tempPa;
	      END_IF;
	    END_IF;
	  END_IF;
	  
	END_REGION ; 
	#LKinCtrl_CalcCircCenterByRadiusAndEndPoint := 0; // o.k.
END_FUNCTION

FUNCTION "LKinCtrl_CalcCircleCircleIntersectionPoint" : Word
TITLE = LKinCtrl_CalcCircleCircleIntersectionPoint
{ S7_Optimized_Access := 'TRUE' }
AUTHOR : 'handling.team.automation@siemens.com'
FAMILY : LKinCtrl
VERSION : 5.0
//Determine the points where 2 circles in a common plane intersect
   VAR_INPUT 
      circleCenterPoint1 : "LKinCtrl_typeCOff3DPoint";   // Center point of first circle
      circleCenterPoint2 : "LKinCtrl_typeCOff3DPoint";   // Center point of second circle
      circleRadius1 : LReal;   // Radius of first circle
      circleRadius2 : LReal;   // Radius of second circle
      pathPlane : Int;   // Path plane: XZ= 0, YZ=1, XY= 2
   END_VAR

   VAR_OUTPUT 
      intersectionPointA : "LKinCtrl_typeCOff3DPoint";   // Intersection point a
      intersectionPointB : "LKinCtrl_typeCOff3DPoint";   // Intersection point b
   END_VAR

   VAR_TEMP 
      tempP02 : LReal;
      tempvDiff : "LKinCtrl_typeCOff3DPoint";
      tempCenterDistance : LReal;
      tempH : LReal;
      tempInterPointOffset : "LKinCtrl_typeCOff3DPoint";
      tempP2 : "LKinCtrl_typeCOff3DPoint";
   END_VAR

   VAR CONSTANT 
      COFF_EPS : LReal := 0.001;   // Internal constant
      ERR_COFF_INVALID_PATH_PLANE : Word := 16#8303;   // Error - invalid path plane
      ERR_COFF_CIRCLES_DO_NOT_INTERSECT : Word := 16#8318;   // Error - no solution - circles don't intersect
      ERR_COFF_ONE_CIRC_CONTAINED_IN_THE_OTHER : Word := 16#8319;   // Error - one circle is contained in the other
      ERR_COFF_CIRCLE_CENTERS_EQUAL : Word := 16#8350;   // Error - circle centers are equal infinite intersections (only internal)
   END_VAR


